REGION Network 38: Sepa Gripper Job Interface [Reloading]
   RUNG wire#powerrail
      Contact( "Unit1.Em7.ControlNodes".sepaGripper."step".action1[421] )
      Coil( "Unit1.Em7.ControlNodes".sepaGripper.jobInterface.reLoadJob4.loadingReady )
   END_RUNG
   RUNG wire#powerrail
      Contact( "Unit1.Em7.ControlNodes".sepaGripper."step".action1[1525] )
      Coil( "Unit1.Em7.ControlNodes".sepaGripper.jobInterface.LoadToJRWinderJob15.loadingReady )
   END_RUNG
   // the same network as SCL:
   "Unit1.Em7.ControlNodes".sepaGripper.jobInterface.reLoadJob4.loadingReady := "Unit1.Em7.ControlNodes".sepaGripper."step".action1[421];
   "Unit1.Em7.ControlNodes".sepaGripper.jobInterface.LoadToJRWinderJob15.loadingReady := "Unit1.Em7.ControlNodes".sepaGripper."step".action1[1525];
END_REGION

REGION Network 39: Sepa Gripper Job Interface [UnReloading]
   RUNG wire#powerrail
      Contact( "Unit1.Em7.ControlNodes".sepaGripper."step".action1[510] )
      Coil( "Unit1.Em7.ControlNodes".sepaGripper.jobInterface.reUnloadJob5.unLoadingReady )
   END_RUNG
   RUNG wire#powerrail
      Contact( #instSepaGripperJellyRollUnGripJob5.jobStatus.active )
      Contact( "Unit1.Em7.ControlNodes".cm.softCam.sepaGripperAxisX.okDisChargePos.inPos )
      Contact( "Unit1.Em7.ControlNodes".cm.softCam.sepaGripperAxisZ.okDisChargePos.inPos )
      Contact( "Unit1.Em7.ControlNodes".cm.softCam.sepaGripperAxisC.okDischargePos.inPos )
      Coil( "Unit1.Em7.ControlNodes".sepaGripper.jobInterface.reUnloadJob5.clampRequest )
   END_RUNG
   RUNG wire#powerrail
      Contact( "Unit1.Em7.ControlNodes".sepaGripper."step".action1[581] )
      Coil( "Unit1.Em7.ControlNodes".sepaGripper.jobInterface.reUnloadJob5.unLoadingDone )
   END_RUNG
   // the same network as SCL:
   "Unit1.Em7.ControlNodes".sepaGripper.jobInterface.reUnloadJob5.unLoadingReady := "Unit1.Em7.ControlNodes".sepaGripper."step".action1[510];
   "Unit1.Em7.ControlNodes".sepaGripper.jobInterface.reUnloadJob5.clampRequest := #instSepaGripperJellyRollUnGripJob5.jobStatus.active AND "Unit1.Em7.ControlNodes".cm.softCam.sepaGripperAxisX.okDisChargePos.inPos AND "Unit1.Em7.ControlNodes".cm.softCam.sepaGripperAxisZ.okDisChargePos.inPos AND "Unit1.Em7.ControlNodes".cm.softCam.sepaGripperAxisC.okDischargePos.inPos;
   "Unit1.Em7.ControlNodes".sepaGripper.jobInterface.reUnloadJob5.unLoadingDone := "Unit1.Em7.ControlNodes".sepaGripper."step".action1[581];
END_REGION

REGION Network 40: [Sepa Gripper Job Interface [UnLoading][BA060]][Unused]
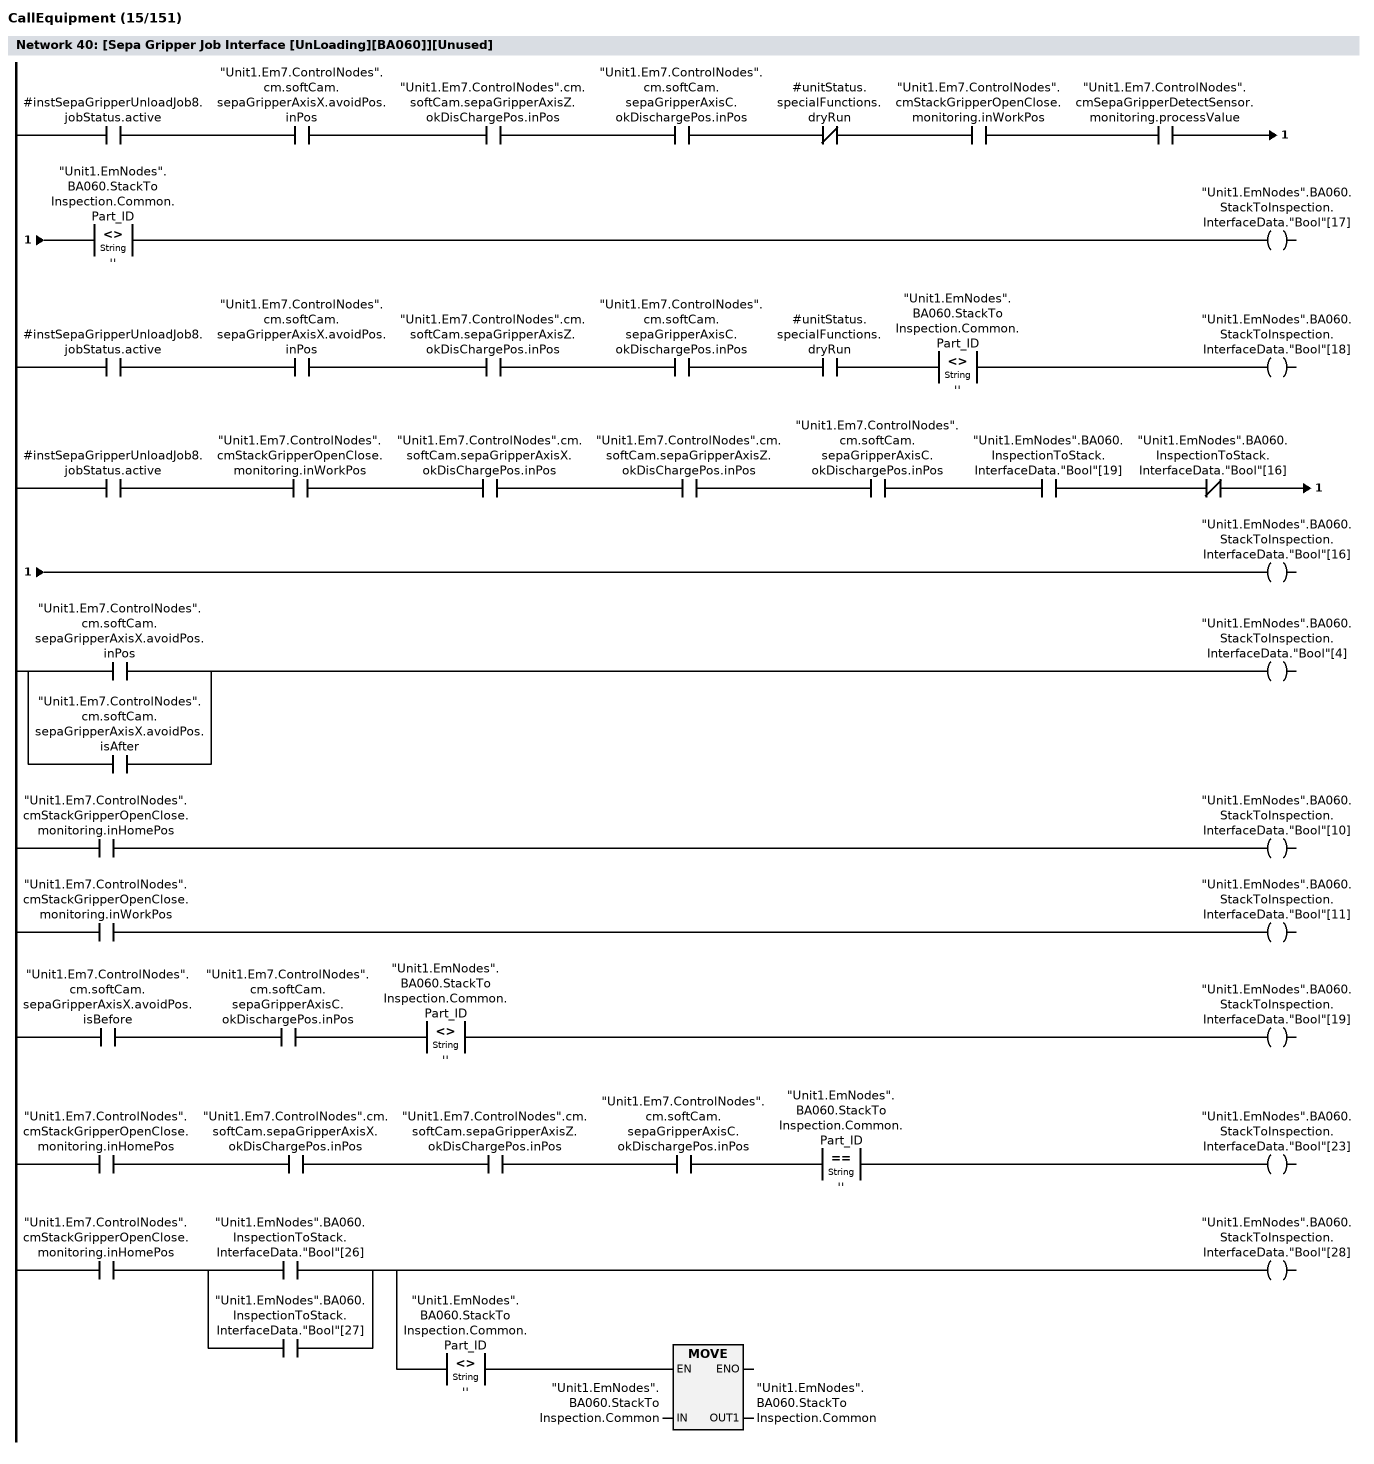
   RUNG wire#powerrail
      Contact( #instSepaGripperUnloadJob8.jobStatus.active )
      Contact( "Unit1.Em7.ControlNodes".cm.softCam.sepaGripperAxisX.avoidPos.inPos )
      Contact( "Unit1.Em7.ControlNodes".cm.softCam.sepaGripperAxisZ.okDisChargePos.inPos )
      Contact( "Unit1.Em7.ControlNodes".cm.softCam.sepaGripperAxisC.okDischargePos.inPos )
      I_Contact( #unitStatus.specialFunctions.dryRun )
      Contact( "Unit1.Em7.ControlNodes".cmStackGripperOpenClose.monitoring.inWorkPos )
      Contact( "Unit1.Em7.ControlNodes".cmSepaGripperDetectSensor.monitoring.processValue )
      { S7_Templates := "SrcType := String" } NE_Contact(in1 := "Unit1.EmNodes".BA060.StackToInspection.Common.Part_ID, in2 := '')
      Coil( "Unit1.EmNodes".BA060.StackToInspection.InterfaceData."Bool"[17] )
   END_RUNG
   RUNG wire#powerrail
      Contact( #instSepaGripperUnloadJob8.jobStatus.active )
      Contact( "Unit1.Em7.ControlNodes".cm.softCam.sepaGripperAxisX.avoidPos.inPos )
      Contact( "Unit1.Em7.ControlNodes".cm.softCam.sepaGripperAxisZ.okDisChargePos.inPos )
      Contact( "Unit1.Em7.ControlNodes".cm.softCam.sepaGripperAxisC.okDischargePos.inPos )
      Contact( #unitStatus.specialFunctions.dryRun )
      { S7_Templates := "SrcType := String" } NE_Contact(in1 := "Unit1.EmNodes".BA060.StackToInspection.Common.Part_ID, in2 := '')
      Coil( "Unit1.EmNodes".BA060.StackToInspection.InterfaceData."Bool"[18] )
   END_RUNG
   RUNG wire#powerrail
      Contact( #instSepaGripperUnloadJob8.jobStatus.active )
      Contact( "Unit1.Em7.ControlNodes".cmStackGripperOpenClose.monitoring.inWorkPos )
      Contact( "Unit1.Em7.ControlNodes".cm.softCam.sepaGripperAxisX.okDisChargePos.inPos )
      Contact( "Unit1.Em7.ControlNodes".cm.softCam.sepaGripperAxisZ.okDisChargePos.inPos )
      Contact( "Unit1.Em7.ControlNodes".cm.softCam.sepaGripperAxisC.okDischargePos.inPos )
      Contact( "Unit1.EmNodes".BA060.InspectionToStack.InterfaceData."Bool"[19] )
      I_Contact( "Unit1.EmNodes".BA060.InspectionToStack.InterfaceData."Bool"[16] )
      Coil( "Unit1.EmNodes".BA060.StackToInspection.InterfaceData."Bool"[16] )
   END_RUNG
   RUNG wire#powerrail
      Contact( "Unit1.Em7.ControlNodes".cm.softCam.sepaGripperAxisX.avoidPos.inPos )
      wire#w1
      Coil( "Unit1.EmNodes".BA060.StackToInspection.InterfaceData."Bool"[4] )
   END_RUNG
   RUNG wire#powerrail
      Contact( "Unit1.Em7.ControlNodes".cm.softCam.sepaGripperAxisX.avoidPos.isAfter )
   END_RUNG wire#w1
   RUNG wire#powerrail
      Contact( "Unit1.Em7.ControlNodes".cmStackGripperOpenClose.monitoring.inHomePos )
      Coil( "Unit1.EmNodes".BA060.StackToInspection.InterfaceData."Bool"[10] )
   END_RUNG
   RUNG wire#powerrail
      Contact( "Unit1.Em7.ControlNodes".cmStackGripperOpenClose.monitoring.inWorkPos )
      Coil( "Unit1.EmNodes".BA060.StackToInspection.InterfaceData."Bool"[11] )
   END_RUNG
   RUNG wire#powerrail
      Contact( "Unit1.Em7.ControlNodes".cm.softCam.sepaGripperAxisX.avoidPos.isBefore )
      Contact( "Unit1.Em7.ControlNodes".cm.softCam.sepaGripperAxisC.okDischargePos.inPos )
      { S7_Templates := "SrcType := String" } NE_Contact(in1 := "Unit1.EmNodes".BA060.StackToInspection.Common.Part_ID, in2 := '')
      Coil( "Unit1.EmNodes".BA060.StackToInspection.InterfaceData."Bool"[19] )
   END_RUNG
   RUNG wire#powerrail
      Contact( "Unit1.Em7.ControlNodes".cmStackGripperOpenClose.monitoring.inHomePos )
      Contact( "Unit1.Em7.ControlNodes".cm.softCam.sepaGripperAxisX.okDisChargePos.inPos )
      Contact( "Unit1.Em7.ControlNodes".cm.softCam.sepaGripperAxisZ.okDisChargePos.inPos )
      Contact( "Unit1.Em7.ControlNodes".cm.softCam.sepaGripperAxisC.okDischargePos.inPos )
      { S7_Templates := "SrcType := String" } EQ_Contact(in1 := "Unit1.EmNodes".BA060.StackToInspection.Common.Part_ID, in2 := '')
      Coil( "Unit1.EmNodes".BA060.StackToInspection.InterfaceData."Bool"[23] )
   END_RUNG
   RUNG wire#powerrail
      Contact( "Unit1.Em7.ControlNodes".cmStackGripperOpenClose.monitoring.inHomePos )
      wire#w2
      Contact( "Unit1.EmNodes".BA060.InspectionToStack.InterfaceData."Bool"[26] )
      wire#w3
      Coil( "Unit1.EmNodes".BA060.StackToInspection.InterfaceData."Bool"[28] )
   END_RUNG
   RUNG wire#w2
      Contact( "Unit1.EmNodes".BA060.InspectionToStack.InterfaceData."Bool"[27] )
   END_RUNG wire#w3
   RUNG wire#w3
      { S7_Templates := "SrcType := String" } NE_Contact(in1 := "Unit1.EmNodes".BA060.StackToInspection.Common.Part_ID, in2 := '')
      Move(in := "Unit1.EmNodes".BA060.StackToInspection.Common, out1 => "Unit1.EmNodes".BA060.StackToInspection.Common)
   END_RUNG
   // the same network as SCL:
   "Unit1.EmNodes".BA060.StackToInspection.InterfaceData."Bool"[17] := #instSepaGripperUnloadJob8.jobStatus.active AND "Unit1.Em7.ControlNodes".cm.softCam.sepaGripperAxisX.avoidPos.inPos AND "Unit1.Em7.ControlNodes".cm.softCam.sepaGripperAxisZ.okDisChargePos.inPos AND "Unit1.Em7.ControlNodes".cm.softCam.sepaGripperAxisC.okDischargePos.inPos AND NOT #unitStatus.specialFunctions.dryRun AND "Unit1.Em7.ControlNodes".cmStackGripperOpenClose.monitoring.inWorkPos AND "Unit1.Em7.ControlNodes".cmSepaGripperDetectSensor.monitoring.processValue AND ("Unit1.EmNodes".BA060.StackToInspection.Common.Part_ID <> '');
   "Unit1.EmNodes".BA060.StackToInspection.InterfaceData."Bool"[18] := #instSepaGripperUnloadJob8.jobStatus.active AND "Unit1.Em7.ControlNodes".cm.softCam.sepaGripperAxisX.avoidPos.inPos AND "Unit1.Em7.ControlNodes".cm.softCam.sepaGripperAxisZ.okDisChargePos.inPos AND "Unit1.Em7.ControlNodes".cm.softCam.sepaGripperAxisC.okDischargePos.inPos AND #unitStatus.specialFunctions.dryRun AND ("Unit1.EmNodes".BA060.StackToInspection.Common.Part_ID <> '');
   "Unit1.EmNodes".BA060.StackToInspection.InterfaceData."Bool"[16] := #instSepaGripperUnloadJob8.jobStatus.active AND "Unit1.Em7.ControlNodes".cmStackGripperOpenClose.monitoring.inWorkPos AND "Unit1.Em7.ControlNodes".cm.softCam.sepaGripperAxisX.okDisChargePos.inPos AND "Unit1.Em7.ControlNodes".cm.softCam.sepaGripperAxisZ.okDisChargePos.inPos AND "Unit1.Em7.ControlNodes".cm.softCam.sepaGripperAxisC.okDischargePos.inPos AND "Unit1.EmNodes".BA060.InspectionToStack.InterfaceData."Bool"[19] AND NOT "Unit1.EmNodes".BA060.InspectionToStack.InterfaceData."Bool"[16];
   "Unit1.EmNodes".BA060.StackToInspection.InterfaceData."Bool"[4] := "Unit1.Em7.ControlNodes".cm.softCam.sepaGripperAxisX.avoidPos.inPos OR "Unit1.Em7.ControlNodes".cm.softCam.sepaGripperAxisX.avoidPos.isAfter;
   "Unit1.EmNodes".BA060.StackToInspection.InterfaceData."Bool"[10] := "Unit1.Em7.ControlNodes".cmStackGripperOpenClose.monitoring.inHomePos;
   "Unit1.EmNodes".BA060.StackToInspection.InterfaceData."Bool"[11] := "Unit1.Em7.ControlNodes".cmStackGripperOpenClose.monitoring.inWorkPos;
   "Unit1.EmNodes".BA060.StackToInspection.InterfaceData."Bool"[19] := "Unit1.Em7.ControlNodes".cm.softCam.sepaGripperAxisX.avoidPos.isBefore AND "Unit1.Em7.ControlNodes".cm.softCam.sepaGripperAxisC.okDischargePos.inPos AND ("Unit1.EmNodes".BA060.StackToInspection.Common.Part_ID <> '');
   "Unit1.EmNodes".BA060.StackToInspection.InterfaceData."Bool"[23] := "Unit1.Em7.ControlNodes".cmStackGripperOpenClose.monitoring.inHomePos AND "Unit1.Em7.ControlNodes".cm.softCam.sepaGripperAxisX.okDisChargePos.inPos AND "Unit1.Em7.ControlNodes".cm.softCam.sepaGripperAxisZ.okDisChargePos.inPos AND "Unit1.Em7.ControlNodes".cm.softCam.sepaGripperAxisC.okDischargePos.inPos AND ("Unit1.EmNodes".BA060.StackToInspection.Common.Part_ID = '');
   "Unit1.EmNodes".BA060.StackToInspection.InterfaceData."Bool"[28] := "Unit1.Em7.ControlNodes".cmStackGripperOpenClose.monitoring.inHomePos AND ("Unit1.EmNodes".BA060.InspectionToStack.InterfaceData."Bool"[26] OR "Unit1.EmNodes".BA060.InspectionToStack.InterfaceData."Bool"[27]);
   IF "Unit1.Em7.ControlNodes".cmStackGripperOpenClose.monitoring.inHomePos AND ("Unit1.EmNodes".BA060.InspectionToStack.InterfaceData."Bool"[26] OR "Unit1.EmNodes".BA060.InspectionToStack.InterfaceData."Bool"[27]) AND ("Unit1.EmNodes".BA060.StackToInspection.Common.Part_ID <> '') THEN
       "Unit1.EmNodes".BA060.StackToInspection.Common := "Unit1.EmNodes".BA060.StackToInspection.Common;
   END_IF;
END_REGION

REGION Network 41: Sepa Gripper Job Interface Working Done
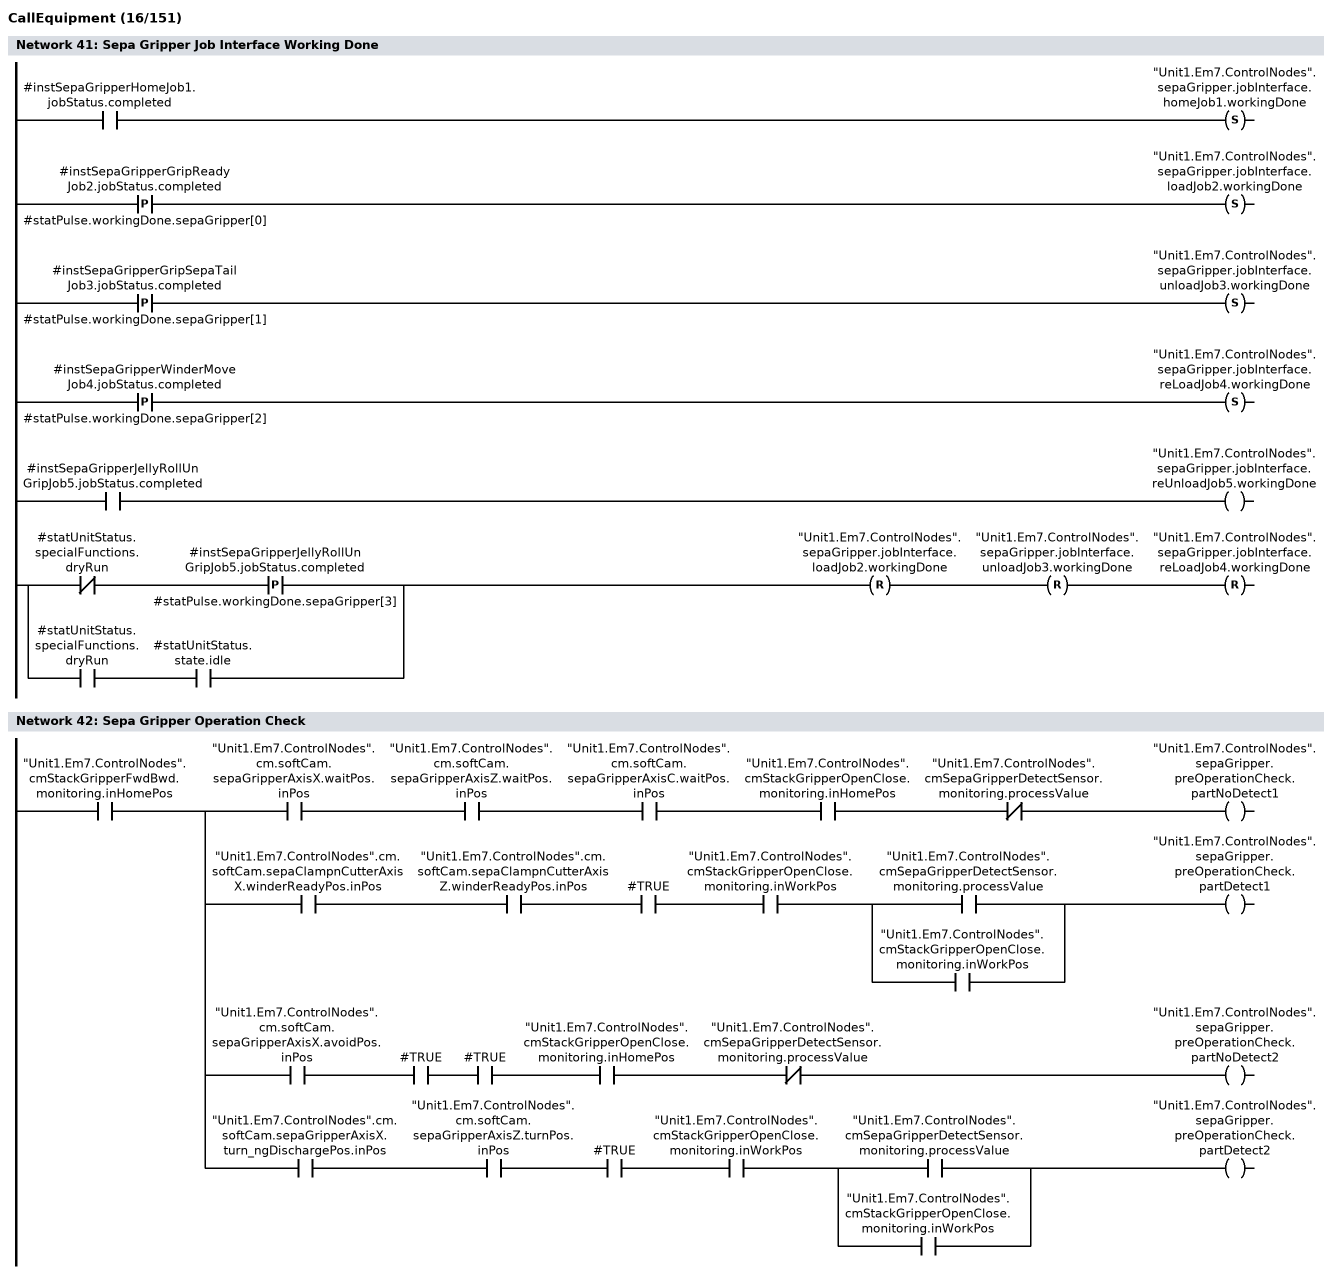
   RUNG wire#powerrail
      Contact( #instSepaGripperHomeJob1.jobStatus.completed )
      S_Coil( "Unit1.Em7.ControlNodes".sepaGripper.jobInterface.homeJob1.workingDone )
   END_RUNG
   RUNG wire#powerrail
      P_Contact(operand := #instSepaGripperGripReadyJob2.jobStatus.completed, bit := #statPulse.workingDone.sepaGripper[0])
      S_Coil( "Unit1.Em7.ControlNodes".sepaGripper.jobInterface.loadJob2.workingDone )
   END_RUNG
   RUNG wire#powerrail
      P_Contact(operand := #instSepaGripperGripSepaTailJob3.jobStatus.completed, bit := #statPulse.workingDone.sepaGripper[1])
      S_Coil( "Unit1.Em7.ControlNodes".sepaGripper.jobInterface.unloadJob3.workingDone )
   END_RUNG
   RUNG wire#powerrail
      P_Contact(operand := #instSepaGripperWinderMoveJob4.jobStatus.completed, bit := #statPulse.workingDone.sepaGripper[2])
      S_Coil( "Unit1.Em7.ControlNodes".sepaGripper.jobInterface.reLoadJob4.workingDone )
   END_RUNG
   RUNG wire#powerrail
      Contact( #instSepaGripperJellyRollUnGripJob5.jobStatus.completed )
      Coil( "Unit1.Em7.ControlNodes".sepaGripper.jobInterface.reUnloadJob5.workingDone )
   END_RUNG
   RUNG wire#powerrail
      I_Contact( #statUnitStatus.specialFunctions.dryRun )
      P_Contact(operand := #instSepaGripperJellyRollUnGripJob5.jobStatus.completed, bit := #statPulse.workingDone.sepaGripper[3])
      wire#w1
      R_Coil( "Unit1.Em7.ControlNodes".sepaGripper.jobInterface.loadJob2.workingDone )
      R_Coil( "Unit1.Em7.ControlNodes".sepaGripper.jobInterface.unloadJob3.workingDone )
      R_Coil( "Unit1.Em7.ControlNodes".sepaGripper.jobInterface.reLoadJob4.workingDone )
   END_RUNG
   RUNG wire#powerrail
      Contact( #statUnitStatus.specialFunctions.dryRun )
      Contact( #statUnitStatus.state.idle )
   END_RUNG wire#w1
   // the same network as SCL:
   IF #instSepaGripperHomeJob1.jobStatus.completed THEN
       "Unit1.Em7.ControlNodes".sepaGripper.jobInterface.homeJob1.workingDone := TRUE;
   END_IF;
   #_w1 := #instSepaGripperGripReadyJob2.jobStatus.completed AND NOT #statPulse.workingDone.sepaGripper[0];   // rising edge of #instSepaGripperGripReadyJob2.jobStatus.completed
   #statPulse.workingDone.sepaGripper[0] := #instSepaGripperGripReadyJob2.jobStatus.completed;
   IF #_w1 THEN "Unit1.Em7.ControlNodes".sepaGripper.jobInterface.loadJob2.workingDone := TRUE; END_IF;
   #_w2 := #instSepaGripperGripSepaTailJob3.jobStatus.completed AND NOT #statPulse.workingDone.sepaGripper[1];   // rising edge of #instSepaGripperGripSepaTailJob3.jobStatus.completed
   #statPulse.workingDone.sepaGripper[1] := #instSepaGripperGripSepaTailJob3.jobStatus.completed;
   IF #_w2 THEN "Unit1.Em7.ControlNodes".sepaGripper.jobInterface.unloadJob3.workingDone := TRUE; END_IF;
   #_w3 := #instSepaGripperWinderMoveJob4.jobStatus.completed AND NOT #statPulse.workingDone.sepaGripper[2];   // rising edge of #instSepaGripperWinderMoveJob4.jobStatus.completed
   #statPulse.workingDone.sepaGripper[2] := #instSepaGripperWinderMoveJob4.jobStatus.completed;
   IF #_w3 THEN "Unit1.Em7.ControlNodes".sepaGripper.jobInterface.reLoadJob4.workingDone := TRUE; END_IF;
   "Unit1.Em7.ControlNodes".sepaGripper.jobInterface.reUnloadJob5.workingDone := #instSepaGripperJellyRollUnGripJob5.jobStatus.completed;
   #_w4 := NOT #statUnitStatus.specialFunctions.dryRun AND #instSepaGripperJellyRollUnGripJob5.jobStatus.completed AND NOT #statPulse.workingDone.sepaGripper[3];   // rising edge of #instSepaGripperJellyRollUnGripJob5.jobStatus.completed
   #statPulse.workingDone.sepaGripper[3] := #instSepaGripperJellyRollUnGripJob5.jobStatus.completed;
   IF #_w4 OR (#statUnitStatus.specialFunctions.dryRun AND #statUnitStatus.state.idle) THEN
       "Unit1.Em7.ControlNodes".sepaGripper.jobInterface.loadJob2.workingDone := FALSE;
       "Unit1.Em7.ControlNodes".sepaGripper.jobInterface.unloadJob3.workingDone := FALSE;
       "Unit1.Em7.ControlNodes".sepaGripper.jobInterface.reLoadJob4.workingDone := FALSE;
   END_IF;
END_REGION

REGION Network 42: Sepa Gripper Operation Check
   RUNG wire#powerrail
      Contact( "Unit1.Em7.ControlNodes".cmStackGripperFwdBwd.monitoring.inHomePos )
      wire#w1
      Contact( "Unit1.Em7.ControlNodes".cm.softCam.sepaGripperAxisX.waitPos.inPos )
      Contact( "Unit1.Em7.ControlNodes".cm.softCam.sepaGripperAxisZ.waitPos.inPos )
      Contact( "Unit1.Em7.ControlNodes".cm.softCam.sepaGripperAxisC.waitPos.inPos )
      Contact( "Unit1.Em7.ControlNodes".cmStackGripperOpenClose.monitoring.inHomePos )
      I_Contact( "Unit1.Em7.ControlNodes".cmSepaGripperDetectSensor.monitoring.processValue )
      Coil( "Unit1.Em7.ControlNodes".sepaGripper.preOperationCheck.partNoDetect1 )
   END_RUNG
   RUNG wire#w1
      Contact( "Unit1.Em7.ControlNodes".cm.softCam.sepaClampnCutterAxisX.winderReadyPos.inPos )
      Contact( "Unit1.Em7.ControlNodes".cm.softCam.sepaClampnCutterAxisZ.winderReadyPos.inPos )
      Contact( #TRUE )
      Contact( "Unit1.Em7.ControlNodes".cmStackGripperOpenClose.monitoring.inWorkPos )
      wire#w2
      Contact( "Unit1.Em7.ControlNodes".cmSepaGripperDetectSensor.monitoring.processValue )
      wire#w3
      Coil( "Unit1.Em7.ControlNodes".sepaGripper.preOperationCheck.partDetect1 )
   END_RUNG
   RUNG wire#w2
      Contact( "Unit1.Em7.ControlNodes".cmStackGripperOpenClose.monitoring.inWorkPos )
   END_RUNG wire#w3
   RUNG wire#w1
      Contact( "Unit1.Em7.ControlNodes".cm.softCam.sepaGripperAxisX.avoidPos.inPos )
      Contact( #TRUE )
      Contact( #TRUE )
      Contact( "Unit1.Em7.ControlNodes".cmStackGripperOpenClose.monitoring.inHomePos )
      I_Contact( "Unit1.Em7.ControlNodes".cmSepaGripperDetectSensor.monitoring.processValue )
      Coil( "Unit1.Em7.ControlNodes".sepaGripper.preOperationCheck.partNoDetect2 )
   END_RUNG
   RUNG wire#w1
      Contact( "Unit1.Em7.ControlNodes".cm.softCam.sepaGripperAxisX.turn_ngDischargePos.inPos )
      Contact( "Unit1.Em7.ControlNodes".cm.softCam.sepaGripperAxisZ.turnPos.inPos )
      Contact( #TRUE )
      Contact( "Unit1.Em7.ControlNodes".cmStackGripperOpenClose.monitoring.inWorkPos )
      wire#w4
      Contact( "Unit1.Em7.ControlNodes".cmSepaGripperDetectSensor.monitoring.processValue )
      wire#w5
      Coil( "Unit1.Em7.ControlNodes".sepaGripper.preOperationCheck.partDetect2 )
   END_RUNG
   RUNG wire#w4
      Contact( "Unit1.Em7.ControlNodes".cmStackGripperOpenClose.monitoring.inWorkPos )
   END_RUNG wire#w5
   // the same network as SCL:
   "Unit1.Em7.ControlNodes".sepaGripper.preOperationCheck.partNoDetect1 := "Unit1.Em7.ControlNodes".cmStackGripperFwdBwd.monitoring.inHomePos AND "Unit1.Em7.ControlNodes".cm.softCam.sepaGripperAxisX.waitPos.inPos AND "Unit1.Em7.ControlNodes".cm.softCam.sepaGripperAxisZ.waitPos.inPos AND "Unit1.Em7.ControlNodes".cm.softCam.sepaGripperAxisC.waitPos.inPos AND "Unit1.Em7.ControlNodes".cmStackGripperOpenClose.monitoring.inHomePos AND NOT "Unit1.Em7.ControlNodes".cmSepaGripperDetectSensor.monitoring.processValue;
   "Unit1.Em7.ControlNodes".sepaGripper.preOperationCheck.partDetect1 := "Unit1.Em7.ControlNodes".cmStackGripperFwdBwd.monitoring.inHomePos AND "Unit1.Em7.ControlNodes".cm.softCam.sepaClampnCutterAxisX.winderReadyPos.inPos AND "Unit1.Em7.ControlNodes".cm.softCam.sepaClampnCutterAxisZ.winderReadyPos.inPos AND #TRUE AND "Unit1.Em7.ControlNodes".cmStackGripperOpenClose.monitoring.inWorkPos AND ("Unit1.Em7.ControlNodes".cmSepaGripperDetectSensor.monitoring.processValue OR "Unit1.Em7.ControlNodes".cmStackGripperOpenClose.monitoring.inWorkPos);
   "Unit1.Em7.ControlNodes".sepaGripper.preOperationCheck.partNoDetect2 := "Unit1.Em7.ControlNodes".cmStackGripperFwdBwd.monitoring.inHomePos AND "Unit1.Em7.ControlNodes".cm.softCam.sepaGripperAxisX.avoidPos.inPos AND #TRUE AND #TRUE AND "Unit1.Em7.ControlNodes".cmStackGripperOpenClose.monitoring.inHomePos AND NOT "Unit1.Em7.ControlNodes".cmSepaGripperDetectSensor.monitoring.processValue;
   "Unit1.Em7.ControlNodes".sepaGripper.preOperationCheck.partDetect2 := "Unit1.Em7.ControlNodes".cmStackGripperFwdBwd.monitoring.inHomePos AND "Unit1.Em7.ControlNodes".cm.softCam.sepaGripperAxisX.turn_ngDischargePos.inPos AND "Unit1.Em7.ControlNodes".cm.softCam.sepaGripperAxisZ.turnPos.inPos AND #TRUE AND "Unit1.Em7.ControlNodes".cmStackGripperOpenClose.monitoring.inWorkPos AND ("Unit1.Em7.ControlNodes".cmSepaGripperDetectSensor.monitoring.processValue OR "Unit1.Em7.ControlNodes".cmStackGripperOpenClose.monitoring.inWorkPos);
END_REGION

REGION Network 43: Sepa Gripper Operation Check [Cam]
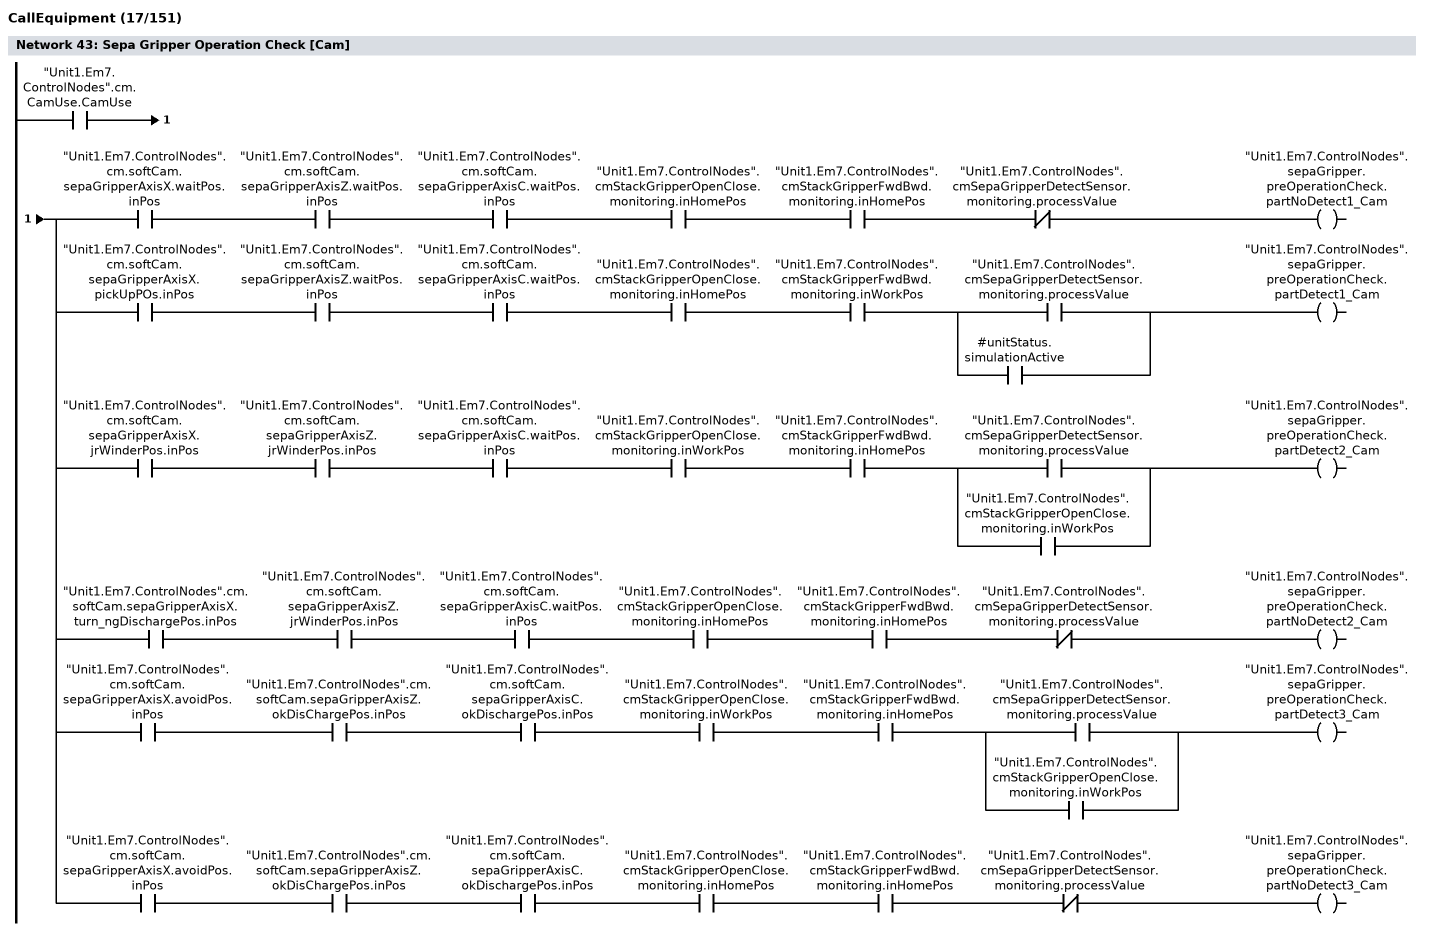
   RUNG wire#powerrail
      Contact( "Unit1.Em7.ControlNodes".cm.CamUse.CamUse )
      wire#w1
      Contact( "Unit1.Em7.ControlNodes".cm.softCam.sepaGripperAxisX.waitPos.inPos )
      Contact( "Unit1.Em7.ControlNodes".cm.softCam.sepaGripperAxisZ.waitPos.inPos )
      Contact( "Unit1.Em7.ControlNodes".cm.softCam.sepaGripperAxisC.waitPos.inPos )
      Contact( "Unit1.Em7.ControlNodes".cmStackGripperOpenClose.monitoring.inHomePos )
      Contact( "Unit1.Em7.ControlNodes".cmStackGripperFwdBwd.monitoring.inHomePos )
      I_Contact( "Unit1.Em7.ControlNodes".cmSepaGripperDetectSensor.monitoring.processValue )
      Coil( "Unit1.Em7.ControlNodes".sepaGripper.preOperationCheck.partNoDetect1_Cam )
   END_RUNG
   RUNG wire#w1
      Contact( "Unit1.Em7.ControlNodes".cm.softCam.sepaGripperAxisX.pickUpPOs.inPos )
      Contact( "Unit1.Em7.ControlNodes".cm.softCam.sepaGripperAxisZ.waitPos.inPos )
      Contact( "Unit1.Em7.ControlNodes".cm.softCam.sepaGripperAxisC.waitPos.inPos )
      Contact( "Unit1.Em7.ControlNodes".cmStackGripperOpenClose.monitoring.inHomePos )
      Contact( "Unit1.Em7.ControlNodes".cmStackGripperFwdBwd.monitoring.inWorkPos )
      wire#w2
      Contact( "Unit1.Em7.ControlNodes".cmSepaGripperDetectSensor.monitoring.processValue )
      wire#w3
      Coil( "Unit1.Em7.ControlNodes".sepaGripper.preOperationCheck.partDetect1_Cam )
   END_RUNG
   RUNG wire#w2
      Contact( #unitStatus.simulationActive )
   END_RUNG wire#w3
   RUNG wire#w1
      Contact( "Unit1.Em7.ControlNodes".cm.softCam.sepaGripperAxisX.jrWinderPos.inPos )
      Contact( "Unit1.Em7.ControlNodes".cm.softCam.sepaGripperAxisZ.jrWinderPos.inPos )
      Contact( "Unit1.Em7.ControlNodes".cm.softCam.sepaGripperAxisC.waitPos.inPos )
      Contact( "Unit1.Em7.ControlNodes".cmStackGripperOpenClose.monitoring.inWorkPos )
      Contact( "Unit1.Em7.ControlNodes".cmStackGripperFwdBwd.monitoring.inHomePos )
      wire#w4
      Contact( "Unit1.Em7.ControlNodes".cmSepaGripperDetectSensor.monitoring.processValue )
      wire#w5
      Coil( "Unit1.Em7.ControlNodes".sepaGripper.preOperationCheck.partDetect2_Cam )
   END_RUNG
   RUNG wire#w4
      Contact( "Unit1.Em7.ControlNodes".cmStackGripperOpenClose.monitoring.inWorkPos )
   END_RUNG wire#w5
   RUNG wire#w1
      Contact( "Unit1.Em7.ControlNodes".cm.softCam.sepaGripperAxisX.turn_ngDischargePos.inPos )
      Contact( "Unit1.Em7.ControlNodes".cm.softCam.sepaGripperAxisZ.jrWinderPos.inPos )
      Contact( "Unit1.Em7.ControlNodes".cm.softCam.sepaGripperAxisC.waitPos.inPos )
      Contact( "Unit1.Em7.ControlNodes".cmStackGripperOpenClose.monitoring.inHomePos )
      Contact( "Unit1.Em7.ControlNodes".cmStackGripperFwdBwd.monitoring.inHomePos )
      I_Contact( "Unit1.Em7.ControlNodes".cmSepaGripperDetectSensor.monitoring.processValue )
      Coil( "Unit1.Em7.ControlNodes".sepaGripper.preOperationCheck.partNoDetect2_Cam )
   END_RUNG
   RUNG wire#w1
      Contact( "Unit1.Em7.ControlNodes".cm.softCam.sepaGripperAxisX.avoidPos.inPos )
      Contact( "Unit1.Em7.ControlNodes".cm.softCam.sepaGripperAxisZ.okDisChargePos.inPos )
      Contact( "Unit1.Em7.ControlNodes".cm.softCam.sepaGripperAxisC.okDischargePos.inPos )
      Contact( "Unit1.Em7.ControlNodes".cmStackGripperOpenClose.monitoring.inWorkPos )
      Contact( "Unit1.Em7.ControlNodes".cmStackGripperFwdBwd.monitoring.inHomePos )
      wire#w6
      Contact( "Unit1.Em7.ControlNodes".cmSepaGripperDetectSensor.monitoring.processValue )
      wire#w7
      Coil( "Unit1.Em7.ControlNodes".sepaGripper.preOperationCheck.partDetect3_Cam )
   END_RUNG
   RUNG wire#w6
      Contact( "Unit1.Em7.ControlNodes".cmStackGripperOpenClose.monitoring.inWorkPos )
   END_RUNG wire#w7
   RUNG wire#w1
      Contact( "Unit1.Em7.ControlNodes".cm.softCam.sepaGripperAxisX.avoidPos.inPos )
      Contact( "Unit1.Em7.ControlNodes".cm.softCam.sepaGripperAxisZ.okDisChargePos.inPos )
      Contact( "Unit1.Em7.ControlNodes".cm.softCam.sepaGripperAxisC.okDischargePos.inPos )
      Contact( "Unit1.Em7.ControlNodes".cmStackGripperOpenClose.monitoring.inHomePos )
      Contact( "Unit1.Em7.ControlNodes".cmStackGripperFwdBwd.monitoring.inHomePos )
      I_Contact( "Unit1.Em7.ControlNodes".cmSepaGripperDetectSensor.monitoring.processValue )
      Coil( "Unit1.Em7.ControlNodes".sepaGripper.preOperationCheck.partNoDetect3_Cam )
   END_RUNG
   // the same network as SCL:
   "Unit1.Em7.ControlNodes".sepaGripper.preOperationCheck.partNoDetect1_Cam := "Unit1.Em7.ControlNodes".cm.CamUse.CamUse AND "Unit1.Em7.ControlNodes".cm.softCam.sepaGripperAxisX.waitPos.inPos AND "Unit1.Em7.ControlNodes".cm.softCam.sepaGripperAxisZ.waitPos.inPos AND "Unit1.Em7.ControlNodes".cm.softCam.sepaGripperAxisC.waitPos.inPos AND "Unit1.Em7.ControlNodes".cmStackGripperOpenClose.monitoring.inHomePos AND "Unit1.Em7.ControlNodes".cmStackGripperFwdBwd.monitoring.inHomePos AND NOT "Unit1.Em7.ControlNodes".cmSepaGripperDetectSensor.monitoring.processValue;
   "Unit1.Em7.ControlNodes".sepaGripper.preOperationCheck.partDetect1_Cam := "Unit1.Em7.ControlNodes".cm.CamUse.CamUse AND "Unit1.Em7.ControlNodes".cm.softCam.sepaGripperAxisX.pickUpPOs.inPos AND "Unit1.Em7.ControlNodes".cm.softCam.sepaGripperAxisZ.waitPos.inPos AND "Unit1.Em7.ControlNodes".cm.softCam.sepaGripperAxisC.waitPos.inPos AND "Unit1.Em7.ControlNodes".cmStackGripperOpenClose.monitoring.inHomePos AND "Unit1.Em7.ControlNodes".cmStackGripperFwdBwd.monitoring.inWorkPos AND ("Unit1.Em7.ControlNodes".cmSepaGripperDetectSensor.monitoring.processValue OR #unitStatus.simulationActive);
   "Unit1.Em7.ControlNodes".sepaGripper.preOperationCheck.partDetect2_Cam := "Unit1.Em7.ControlNodes".cm.CamUse.CamUse AND "Unit1.Em7.ControlNodes".cm.softCam.sepaGripperAxisX.jrWinderPos.inPos AND "Unit1.Em7.ControlNodes".cm.softCam.sepaGripperAxisZ.jrWinderPos.inPos AND "Unit1.Em7.ControlNodes".cm.softCam.sepaGripperAxisC.waitPos.inPos AND "Unit1.Em7.ControlNodes".cmStackGripperOpenClose.monitoring.inWorkPos AND "Unit1.Em7.ControlNodes".cmStackGripperFwdBwd.monitoring.inHomePos AND ("Unit1.Em7.ControlNodes".cmSepaGripperDetectSensor.monitoring.processValue OR "Unit1.Em7.ControlNodes".cmStackGripperOpenClose.monitoring.inWorkPos);
   "Unit1.Em7.ControlNodes".sepaGripper.preOperationCheck.partNoDetect2_Cam := "Unit1.Em7.ControlNodes".cm.CamUse.CamUse AND "Unit1.Em7.ControlNodes".cm.softCam.sepaGripperAxisX.turn_ngDischargePos.inPos AND "Unit1.Em7.ControlNodes".cm.softCam.sepaGripperAxisZ.jrWinderPos.inPos AND "Unit1.Em7.ControlNodes".cm.softCam.sepaGripperAxisC.waitPos.inPos AND "Unit1.Em7.ControlNodes".cmStackGripperOpenClose.monitoring.inHomePos AND "Unit1.Em7.ControlNodes".cmStackGripperFwdBwd.monitoring.inHomePos AND NOT "Unit1.Em7.ControlNodes".cmSepaGripperDetectSensor.monitoring.processValue;
   "Unit1.Em7.ControlNodes".sepaGripper.preOperationCheck.partDetect3_Cam := "Unit1.Em7.ControlNodes".cm.CamUse.CamUse AND "Unit1.Em7.ControlNodes".cm.softCam.sepaGripperAxisX.avoidPos.inPos AND "Unit1.Em7.ControlNodes".cm.softCam.sepaGripperAxisZ.okDisChargePos.inPos AND "Unit1.Em7.ControlNodes".cm.softCam.sepaGripperAxisC.okDischargePos.inPos AND "Unit1.Em7.ControlNodes".cmStackGripperOpenClose.monitoring.inWorkPos AND "Unit1.Em7.ControlNodes".cmStackGripperFwdBwd.monitoring.inHomePos AND ("Unit1.Em7.ControlNodes".cmSepaGripperDetectSensor.monitoring.processValue OR "Unit1.Em7.ControlNodes".cmStackGripperOpenClose.monitoring.inWorkPos);
   "Unit1.Em7.ControlNodes".sepaGripper.preOperationCheck.partNoDetect3_Cam := "Unit1.Em7.ControlNodes".cm.CamUse.CamUse AND "Unit1.Em7.ControlNodes".cm.softCam.sepaGripperAxisX.avoidPos.inPos AND "Unit1.Em7.ControlNodes".cm.softCam.sepaGripperAxisZ.okDisChargePos.inPos AND "Unit1.Em7.ControlNodes".cm.softCam.sepaGripperAxisC.okDischargePos.inPos AND "Unit1.Em7.ControlNodes".cmStackGripperOpenClose.monitoring.inHomePos AND "Unit1.Em7.ControlNodes".cmStackGripperFwdBwd.monitoring.inHomePos AND NOT "Unit1.Em7.ControlNodes".cmSepaGripperDetectSensor.monitoring.processValue;
END_REGION

REGION Network 45: JR Winder Select Job
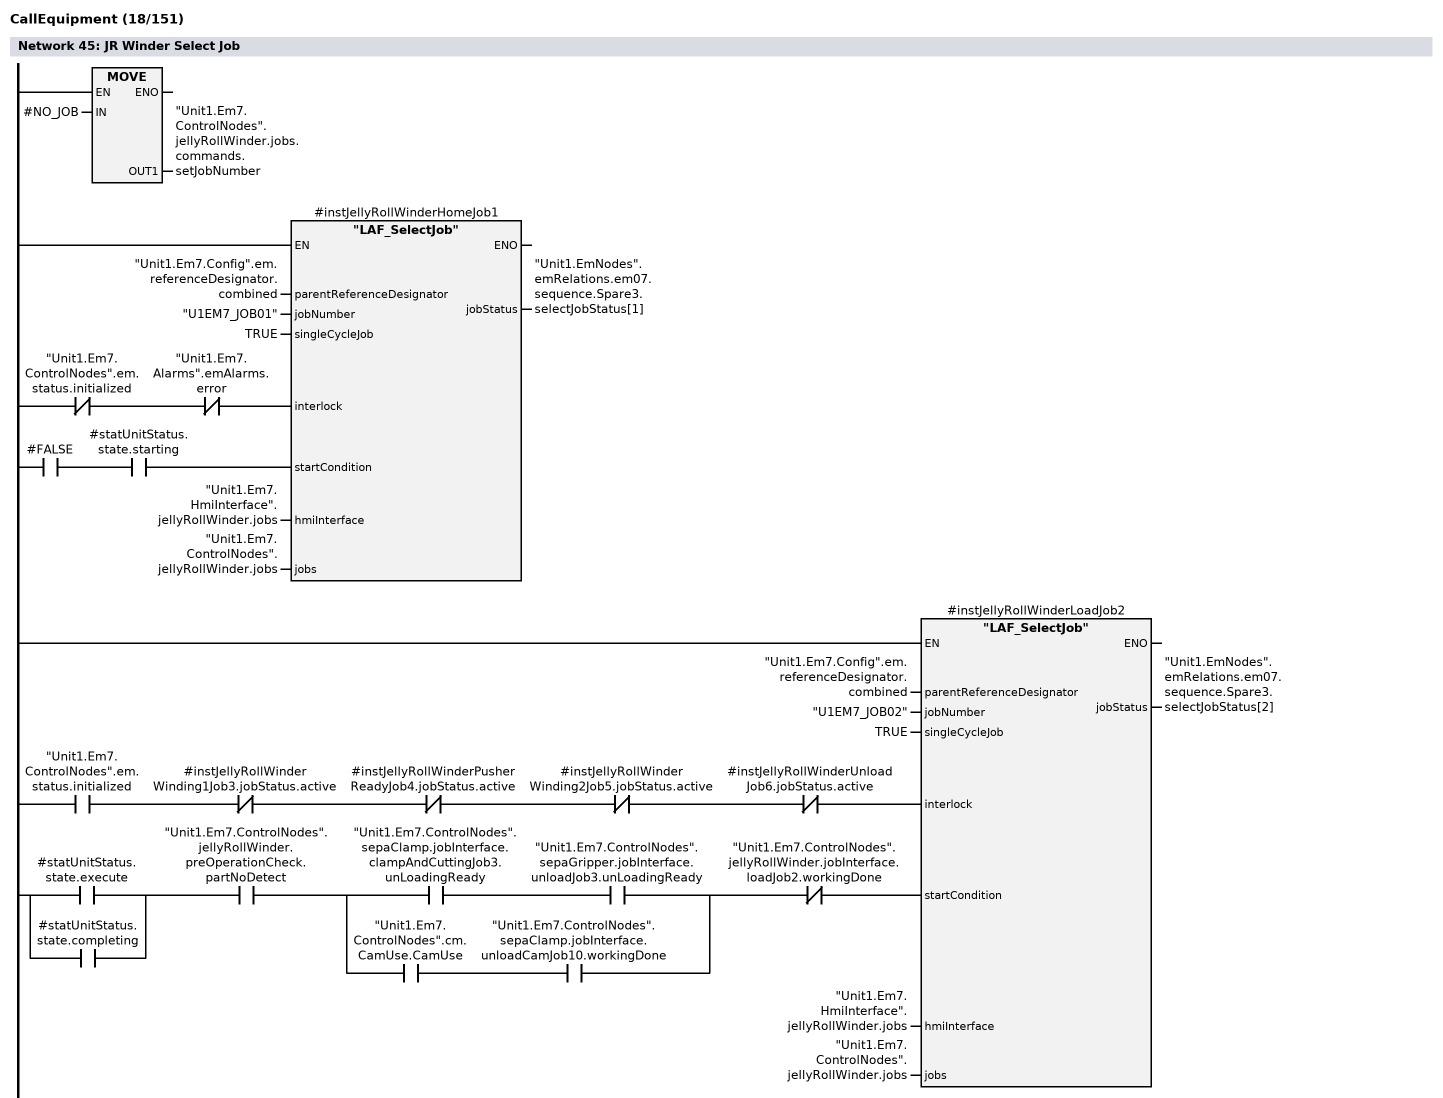
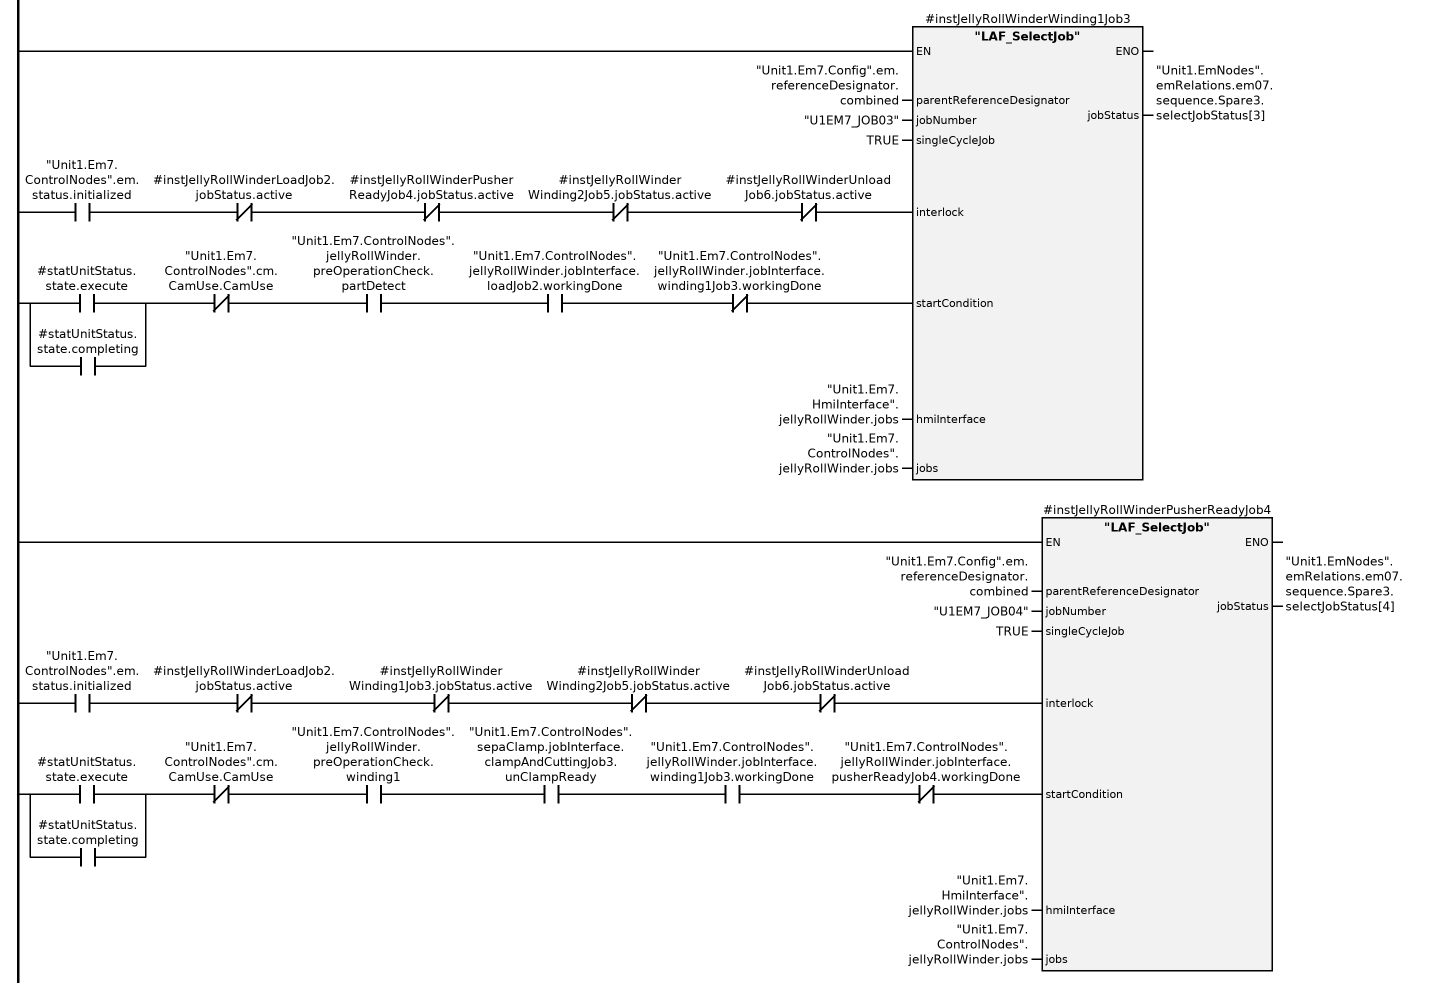
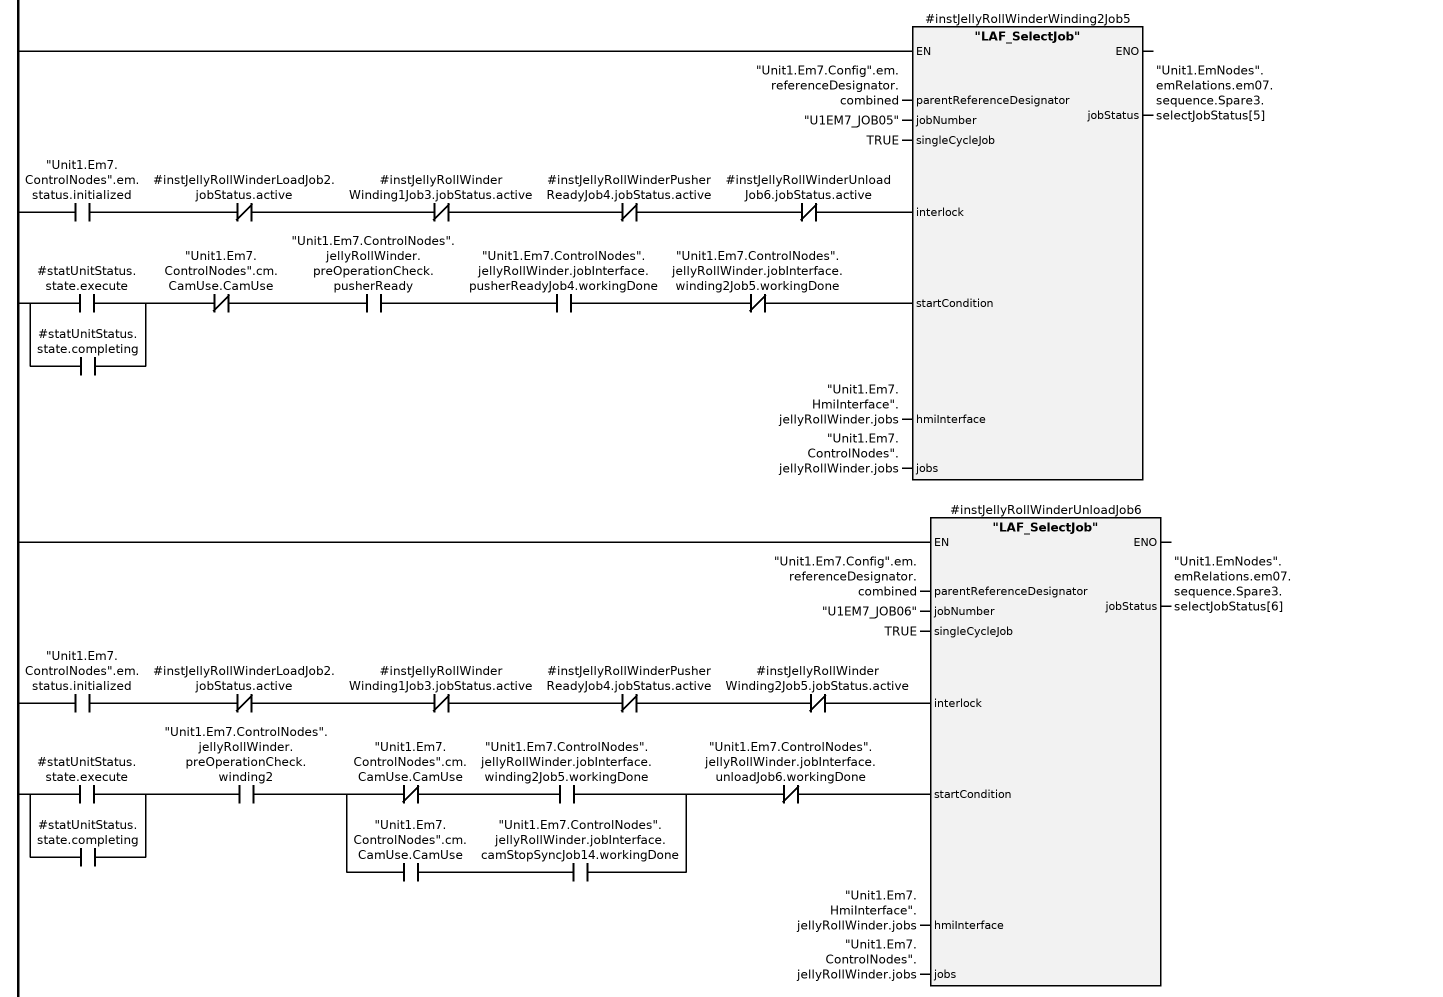
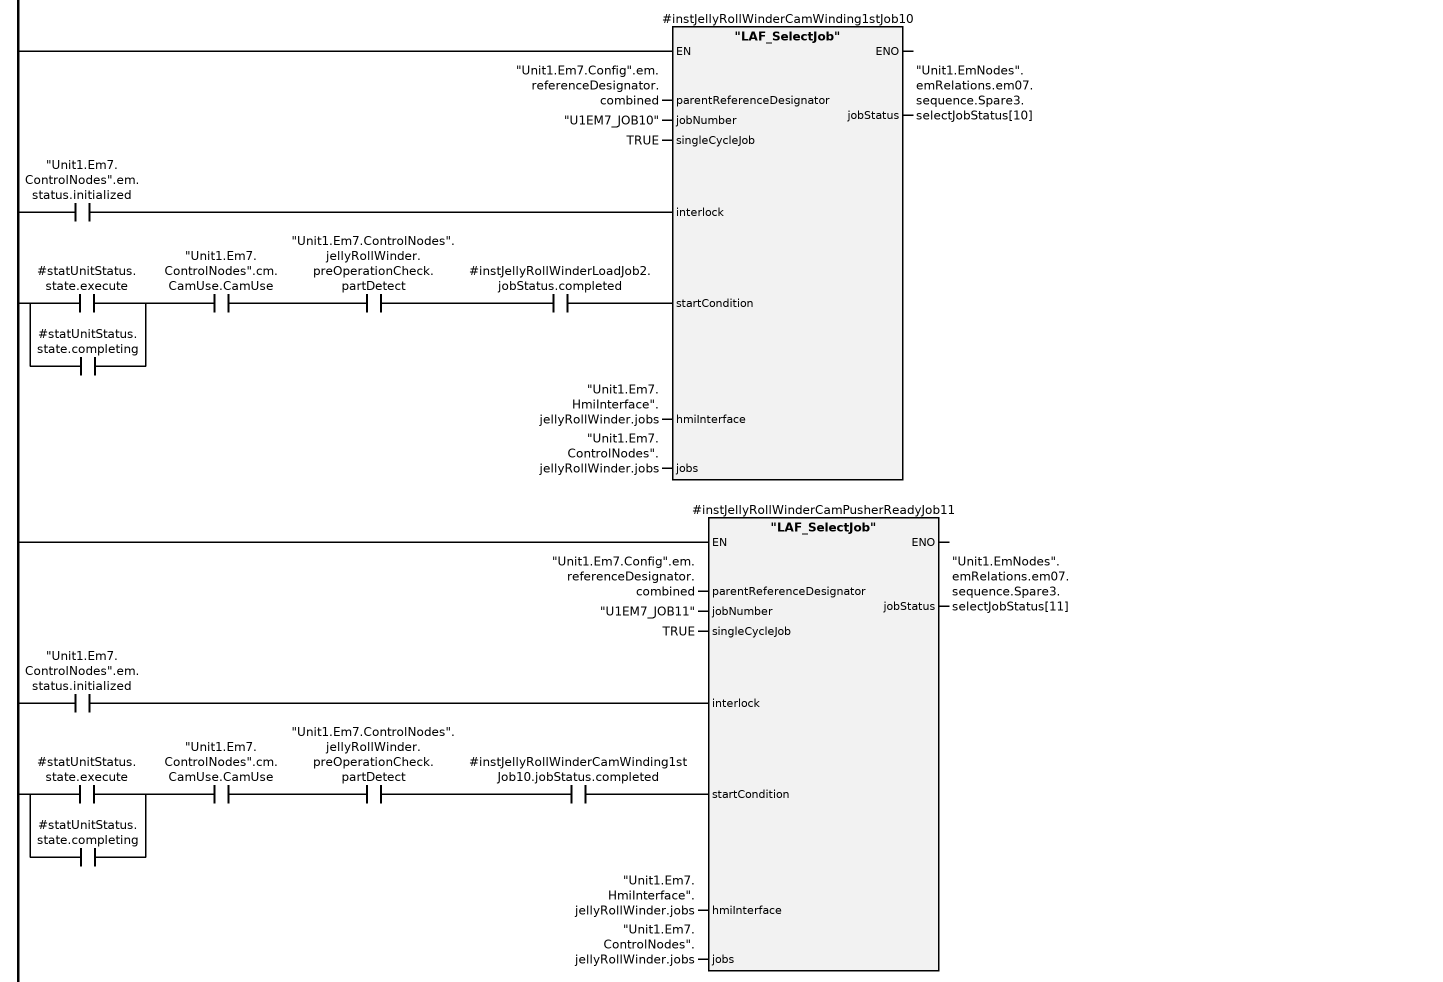
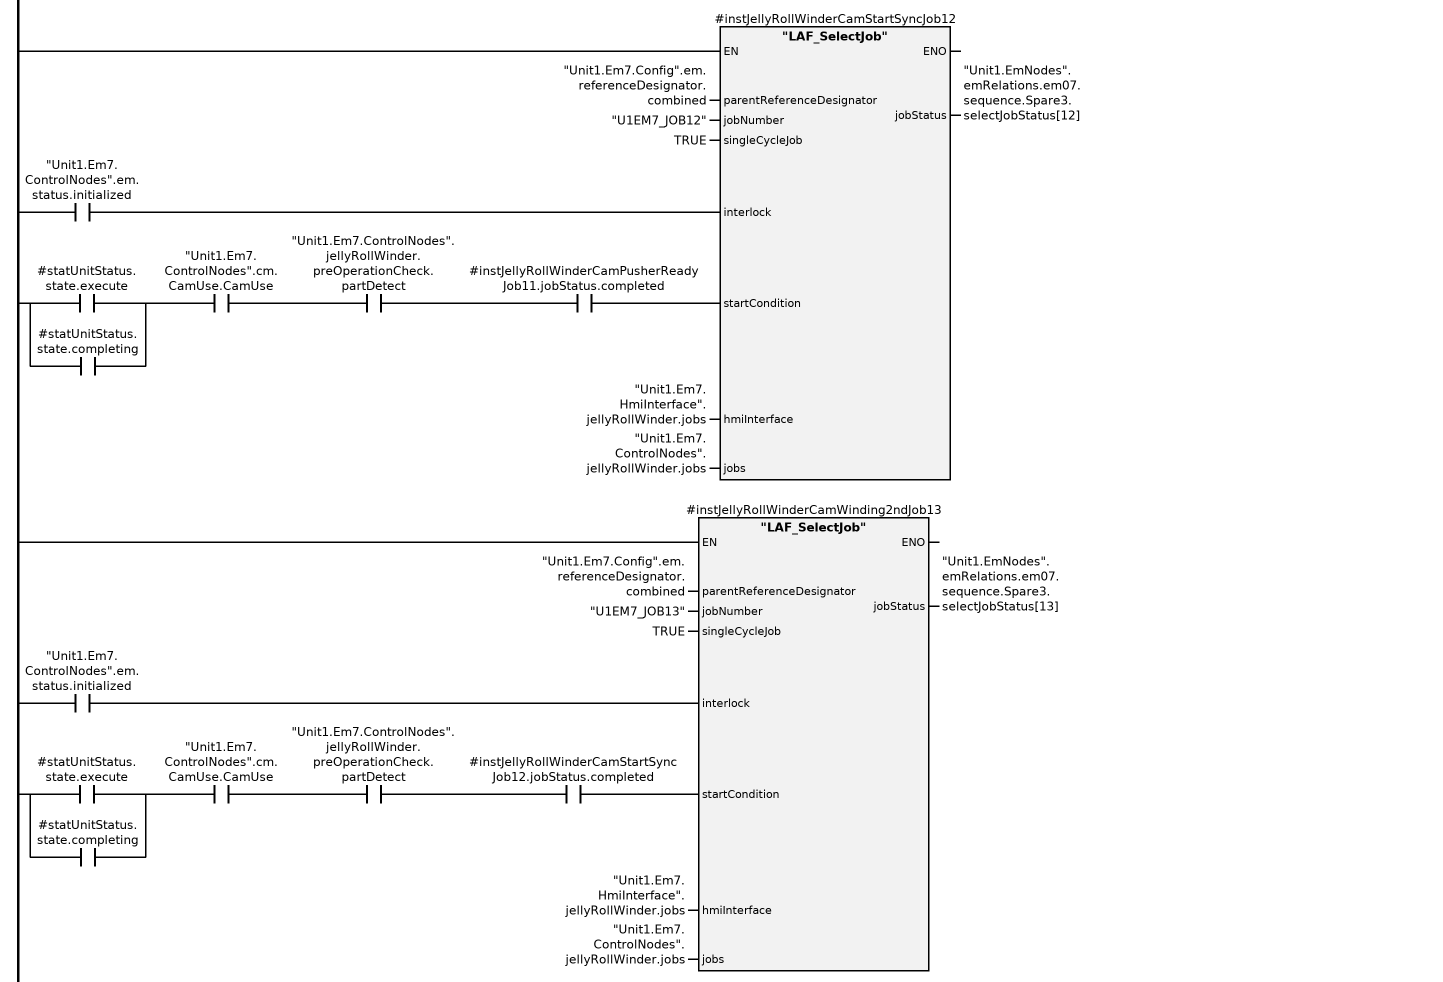
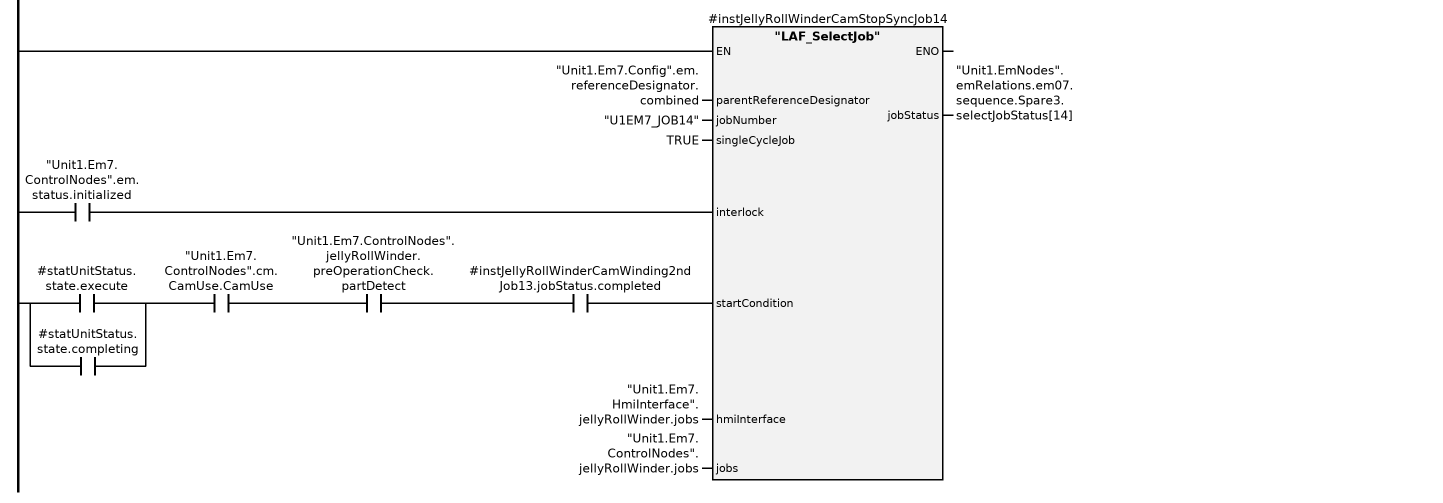
   RUNG wire#powerrail
      Move(in := #NO_JOB, out1 => "Unit1.Em7.ControlNodes".jellyRollWinder.jobs.commands.setJobNumber)
   END_RUNG
   RUNG wire#powerrail
      #instJellyRollWinderHomeJob1(interlock := wire#w1, startCondition := wire#w2, parentReferenceDesignator := "Unit1.Em7.Config".em.referenceDesignator.combined, jobNumber := "U1EM7_JOB01", singleCycleJob := TRUE, hmiInterface := "Unit1.Em7.HmiInterface".jellyRollWinder.jobs, jobs := "Unit1.Em7.ControlNodes".jellyRollWinder.jobs, jobStatus => "Unit1.EmNodes".emRelations.em07.sequence.Spare3.selectJobStatus[1])
   END_RUNG
   RUNG wire#powerrail
      I_Contact( "Unit1.Em7.ControlNodes".em.status.initialized )
      I_Contact( "Unit1.Em7.Alarms".emAlarms.error )
   END_RUNG wire#w1
   RUNG wire#powerrail
      Contact( #FALSE )
      Contact( #statUnitStatus.state.starting )
   END_RUNG wire#w2
   RUNG wire#powerrail
      #instJellyRollWinderLoadJob2(interlock := wire#w3, startCondition := wire#w7, parentReferenceDesignator := "Unit1.Em7.Config".em.referenceDesignator.combined, jobNumber := "U1EM7_JOB02", singleCycleJob := TRUE, hmiInterface := "Unit1.Em7.HmiInterface".jellyRollWinder.jobs, jobs := "Unit1.Em7.ControlNodes".jellyRollWinder.jobs, jobStatus => "Unit1.EmNodes".emRelations.em07.sequence.Spare3.selectJobStatus[2])
   END_RUNG
   RUNG wire#powerrail
      Contact( "Unit1.Em7.ControlNodes".em.status.initialized )
      I_Contact( #instJellyRollWinderWinding1Job3.jobStatus.active )
      I_Contact( #instJellyRollWinderPusherReadyJob4.jobStatus.active )
      I_Contact( #instJellyRollWinderWinding2Job5.jobStatus.active )
      I_Contact( #instJellyRollWinderUnloadJob6.jobStatus.active )
   END_RUNG wire#w3
   RUNG wire#powerrail
      Contact( #statUnitStatus.state.execute )
      wire#w4
      Contact( "Unit1.Em7.ControlNodes".jellyRollWinder.preOperationCheck.partNoDetect )
      wire#w5
      Contact( "Unit1.Em7.ControlNodes".sepaClamp.jobInterface.clampAndCuttingJob3.unLoadingReady )
      Contact( "Unit1.Em7.ControlNodes".sepaGripper.jobInterface.unloadJob3.unLoadingReady )
      wire#w6
      I_Contact( "Unit1.Em7.ControlNodes".jellyRollWinder.jobInterface.loadJob2.workingDone )
   END_RUNG wire#w7
   RUNG wire#powerrail
      Contact( #statUnitStatus.state.completing )
   END_RUNG wire#w4
   RUNG wire#w5
      Contact( "Unit1.Em7.ControlNodes".cm.CamUse.CamUse )
      Contact( "Unit1.Em7.ControlNodes".sepaClamp.jobInterface.unloadCamJob10.workingDone )
   END_RUNG wire#w6
   RUNG wire#powerrail
      #instJellyRollWinderWinding1Job3(interlock := wire#w8, startCondition := wire#w10, parentReferenceDesignator := "Unit1.Em7.Config".em.referenceDesignator.combined, jobNumber := "U1EM7_JOB03", singleCycleJob := TRUE, hmiInterface := "Unit1.Em7.HmiInterface".jellyRollWinder.jobs, jobs := "Unit1.Em7.ControlNodes".jellyRollWinder.jobs, jobStatus => "Unit1.EmNodes".emRelations.em07.sequence.Spare3.selectJobStatus[3])
   END_RUNG
   RUNG wire#powerrail
      Contact( "Unit1.Em7.ControlNodes".em.status.initialized )
      I_Contact( #instJellyRollWinderLoadJob2.jobStatus.active )
      I_Contact( #instJellyRollWinderPusherReadyJob4.jobStatus.active )
      I_Contact( #instJellyRollWinderWinding2Job5.jobStatus.active )
      I_Contact( #instJellyRollWinderUnloadJob6.jobStatus.active )
   END_RUNG wire#w8
   RUNG wire#powerrail
      Contact( #statUnitStatus.state.execute )
      wire#w9
      I_Contact( "Unit1.Em7.ControlNodes".cm.CamUse.CamUse )
      Contact( "Unit1.Em7.ControlNodes".jellyRollWinder.preOperationCheck.partDetect )
      Contact( "Unit1.Em7.ControlNodes".jellyRollWinder.jobInterface.loadJob2.workingDone )
      I_Contact( "Unit1.Em7.ControlNodes".jellyRollWinder.jobInterface.winding1Job3.workingDone )
   END_RUNG wire#w10
   RUNG wire#powerrail
      Contact( #statUnitStatus.state.completing )
   END_RUNG wire#w9
   RUNG wire#powerrail
      #instJellyRollWinderPusherReadyJob4(interlock := wire#w11, startCondition := wire#w13, parentReferenceDesignator := "Unit1.Em7.Config".em.referenceDesignator.combined, jobNumber := "U1EM7_JOB04", singleCycleJob := TRUE, hmiInterface := "Unit1.Em7.HmiInterface".jellyRollWinder.jobs, jobs := "Unit1.Em7.ControlNodes".jellyRollWinder.jobs, jobStatus => "Unit1.EmNodes".emRelations.em07.sequence.Spare3.selectJobStatus[4])
   END_RUNG
   RUNG wire#powerrail
      Contact( "Unit1.Em7.ControlNodes".em.status.initialized )
      I_Contact( #instJellyRollWinderLoadJob2.jobStatus.active )
      I_Contact( #instJellyRollWinderWinding1Job3.jobStatus.active )
      I_Contact( #instJellyRollWinderWinding2Job5.jobStatus.active )
      I_Contact( #instJellyRollWinderUnloadJob6.jobStatus.active )
   END_RUNG wire#w11
   RUNG wire#powerrail
      Contact( #statUnitStatus.state.execute )
      wire#w12
      I_Contact( "Unit1.Em7.ControlNodes".cm.CamUse.CamUse )
      Contact( "Unit1.Em7.ControlNodes".jellyRollWinder.preOperationCheck.winding1 )
      Contact( "Unit1.Em7.ControlNodes".sepaClamp.jobInterface.clampAndCuttingJob3.unClampReady )
      Contact( "Unit1.Em7.ControlNodes".jellyRollWinder.jobInterface.winding1Job3.workingDone )
      I_Contact( "Unit1.Em7.ControlNodes".jellyRollWinder.jobInterface.pusherReadyJob4.workingDone )
   END_RUNG wire#w13
   RUNG wire#powerrail
      Contact( #statUnitStatus.state.completing )
   END_RUNG wire#w12
   RUNG wire#powerrail
      #instJellyRollWinderWinding2Job5(interlock := wire#w14, startCondition := wire#w16, parentReferenceDesignator := "Unit1.Em7.Config".em.referenceDesignator.combined, jobNumber := "U1EM7_JOB05", singleCycleJob := TRUE, hmiInterface := "Unit1.Em7.HmiInterface".jellyRollWinder.jobs, jobs := "Unit1.Em7.ControlNodes".jellyRollWinder.jobs, jobStatus => "Unit1.EmNodes".emRelations.em07.sequence.Spare3.selectJobStatus[5])
   END_RUNG
   RUNG wire#powerrail
      Contact( "Unit1.Em7.ControlNodes".em.status.initialized )
      I_Contact( #instJellyRollWinderLoadJob2.jobStatus.active )
      I_Contact( #instJellyRollWinderWinding1Job3.jobStatus.active )
      I_Contact( #instJellyRollWinderPusherReadyJob4.jobStatus.active )
      I_Contact( #instJellyRollWinderUnloadJob6.jobStatus.active )
   END_RUNG wire#w14
   RUNG wire#powerrail
      Contact( #statUnitStatus.state.execute )
      wire#w15
      I_Contact( "Unit1.Em7.ControlNodes".cm.CamUse.CamUse )
      Contact( "Unit1.Em7.ControlNodes".jellyRollWinder.preOperationCheck.pusherReady )
      Contact( "Unit1.Em7.ControlNodes".jellyRollWinder.jobInterface.pusherReadyJob4.workingDone )
      I_Contact( "Unit1.Em7.ControlNodes".jellyRollWinder.jobInterface.winding2Job5.workingDone )
   END_RUNG wire#w16
   RUNG wire#powerrail
      Contact( #statUnitStatus.state.completing )
   END_RUNG wire#w15
   RUNG wire#powerrail
      #instJellyRollWinderUnloadJob6(interlock := wire#w17, startCondition := wire#w21, parentReferenceDesignator := "Unit1.Em7.Config".em.referenceDesignator.combined, jobNumber := "U1EM7_JOB06", singleCycleJob := TRUE, hmiInterface := "Unit1.Em7.HmiInterface".jellyRollWinder.jobs, jobs := "Unit1.Em7.ControlNodes".jellyRollWinder.jobs, jobStatus => "Unit1.EmNodes".emRelations.em07.sequence.Spare3.selectJobStatus[6])
   END_RUNG
   RUNG wire#powerrail
      Contact( "Unit1.Em7.ControlNodes".em.status.initialized )
      I_Contact( #instJellyRollWinderLoadJob2.jobStatus.active )
      I_Contact( #instJellyRollWinderWinding1Job3.jobStatus.active )
      I_Contact( #instJellyRollWinderPusherReadyJob4.jobStatus.active )
      I_Contact( #instJellyRollWinderWinding2Job5.jobStatus.active )
   END_RUNG wire#w17
   RUNG wire#powerrail
      Contact( #statUnitStatus.state.execute )
      wire#w18
      Contact( "Unit1.Em7.ControlNodes".jellyRollWinder.preOperationCheck.winding2 )
      wire#w19
      I_Contact( "Unit1.Em7.ControlNodes".cm.CamUse.CamUse )
      Contact( "Unit1.Em7.ControlNodes".jellyRollWinder.jobInterface.winding2Job5.workingDone )
      wire#w20
      I_Contact( "Unit1.Em7.ControlNodes".jellyRollWinder.jobInterface.unloadJob6.workingDone )
   END_RUNG wire#w21
   RUNG wire#powerrail
      Contact( #statUnitStatus.state.completing )
   END_RUNG wire#w18
   RUNG wire#w19
      Contact( "Unit1.Em7.ControlNodes".cm.CamUse.CamUse )
      Contact( "Unit1.Em7.ControlNodes".jellyRollWinder.jobInterface.camStopSyncJob14.workingDone )
   END_RUNG wire#w20
   RUNG wire#powerrail
      #instJellyRollWinderCamWinding1stJob10(interlock := wire#w22, startCondition := wire#w24, parentReferenceDesignator := "Unit1.Em7.Config".em.referenceDesignator.combined, jobNumber := "U1EM7_JOB10", singleCycleJob := TRUE, hmiInterface := "Unit1.Em7.HmiInterface".jellyRollWinder.jobs, jobs := "Unit1.Em7.ControlNodes".jellyRollWinder.jobs, jobStatus => "Unit1.EmNodes".emRelations.em07.sequence.Spare3.selectJobStatus[10])
   END_RUNG
   RUNG wire#powerrail
      Contact( "Unit1.Em7.ControlNodes".em.status.initialized )
   END_RUNG wire#w22
   RUNG wire#powerrail
      Contact( #statUnitStatus.state.execute )
      wire#w23
      Contact( "Unit1.Em7.ControlNodes".cm.CamUse.CamUse )
      Contact( "Unit1.Em7.ControlNodes".jellyRollWinder.preOperationCheck.partDetect )
      Contact( #instJellyRollWinderLoadJob2.jobStatus.completed )
   END_RUNG wire#w24
   RUNG wire#powerrail
      Contact( #statUnitStatus.state.completing )
   END_RUNG wire#w23
   RUNG wire#powerrail
      #instJellyRollWinderCamPusherReadyJob11(interlock := wire#w25, startCondition := wire#w27, parentReferenceDesignator := "Unit1.Em7.Config".em.referenceDesignator.combined, jobNumber := "U1EM7_JOB11", singleCycleJob := TRUE, hmiInterface := "Unit1.Em7.HmiInterface".jellyRollWinder.jobs, jobs := "Unit1.Em7.ControlNodes".jellyRollWinder.jobs, jobStatus => "Unit1.EmNodes".emRelations.em07.sequence.Spare3.selectJobStatus[11])
   END_RUNG
   RUNG wire#powerrail
      Contact( "Unit1.Em7.ControlNodes".em.status.initialized )
   END_RUNG wire#w25
   RUNG wire#powerrail
      Contact( #statUnitStatus.state.execute )
      wire#w26
      Contact( "Unit1.Em7.ControlNodes".cm.CamUse.CamUse )
      Contact( "Unit1.Em7.ControlNodes".jellyRollWinder.preOperationCheck.partDetect )
      Contact( #instJellyRollWinderCamWinding1stJob10.jobStatus.completed )
   END_RUNG wire#w27
   RUNG wire#powerrail
      Contact( #statUnitStatus.state.completing )
   END_RUNG wire#w26
   RUNG wire#powerrail
      #instJellyRollWinderCamStartSyncJob12(interlock := wire#w28, startCondition := wire#w30, parentReferenceDesignator := "Unit1.Em7.Config".em.referenceDesignator.combined, jobNumber := "U1EM7_JOB12", singleCycleJob := TRUE, hmiInterface := "Unit1.Em7.HmiInterface".jellyRollWinder.jobs, jobs := "Unit1.Em7.ControlNodes".jellyRollWinder.jobs, jobStatus => "Unit1.EmNodes".emRelations.em07.sequence.Spare3.selectJobStatus[12])
   END_RUNG
   RUNG wire#powerrail
      Contact( "Unit1.Em7.ControlNodes".em.status.initialized )
   END_RUNG wire#w28
   RUNG wire#powerrail
      Contact( #statUnitStatus.state.execute )
      wire#w29
      Contact( "Unit1.Em7.ControlNodes".cm.CamUse.CamUse )
      Contact( "Unit1.Em7.ControlNodes".jellyRollWinder.preOperationCheck.partDetect )
      Contact( #instJellyRollWinderCamPusherReadyJob11.jobStatus.completed )
   END_RUNG wire#w30
   RUNG wire#powerrail
      Contact( #statUnitStatus.state.completing )
   END_RUNG wire#w29
   RUNG wire#powerrail
      #instJellyRollWinderCamWinding2ndJob13(interlock := wire#w31, startCondition := wire#w33, parentReferenceDesignator := "Unit1.Em7.Config".em.referenceDesignator.combined, jobNumber := "U1EM7_JOB13", singleCycleJob := TRUE, hmiInterface := "Unit1.Em7.HmiInterface".jellyRollWinder.jobs, jobs := "Unit1.Em7.ControlNodes".jellyRollWinder.jobs, jobStatus => "Unit1.EmNodes".emRelations.em07.sequence.Spare3.selectJobStatus[13])
   END_RUNG
   RUNG wire#powerrail
      Contact( "Unit1.Em7.ControlNodes".em.status.initialized )
   END_RUNG wire#w31
   RUNG wire#powerrail
      Contact( #statUnitStatus.state.execute )
      wire#w32
      Contact( "Unit1.Em7.ControlNodes".cm.CamUse.CamUse )
      Contact( "Unit1.Em7.ControlNodes".jellyRollWinder.preOperationCheck.partDetect )
      Contact( #instJellyRollWinderCamStartSyncJob12.jobStatus.completed )
   END_RUNG wire#w33
   RUNG wire#powerrail
      Contact( #statUnitStatus.state.completing )
   END_RUNG wire#w32
   RUNG wire#powerrail
      #instJellyRollWinderCamStopSyncJob14(interlock := wire#w34, startCondition := wire#w36, parentReferenceDesignator := "Unit1.Em7.Config".em.referenceDesignator.combined, jobNumber := "U1EM7_JOB14", singleCycleJob := TRUE, hmiInterface := "Unit1.Em7.HmiInterface".jellyRollWinder.jobs, jobs := "Unit1.Em7.ControlNodes".jellyRollWinder.jobs, jobStatus => "Unit1.EmNodes".emRelations.em07.sequence.Spare3.selectJobStatus[14])
   END_RUNG
   RUNG wire#powerrail
      Contact( "Unit1.Em7.ControlNodes".em.status.initialized )
   END_RUNG wire#w34
   RUNG wire#powerrail
      Contact( #statUnitStatus.state.execute )
      wire#w35
      Contact( "Unit1.Em7.ControlNodes".cm.CamUse.CamUse )
      Contact( "Unit1.Em7.ControlNodes".jellyRollWinder.preOperationCheck.partDetect )
      Contact( #instJellyRollWinderCamWinding2ndJob13.jobStatus.completed )
   END_RUNG wire#w36
   RUNG wire#powerrail
      Contact( #statUnitStatus.state.completing )
   END_RUNG wire#w35
   // the same network as SCL:
   "Unit1.Em7.ControlNodes".jellyRollWinder.jobs.commands.setJobNumber := #NO_JOB;
   #instJellyRollWinderHomeJob1(parentReferenceDesignator := "Unit1.Em7.Config".em.referenceDesignator.combined,   // "LAF_SelectJob"
                           jobNumber := "U1EM7_JOB01",
                           singleCycleJob := TRUE,
                           interlock := NOT "Unit1.Em7.ControlNodes".em.status.initialized AND NOT "Unit1.Em7.Alarms".emAlarms.error,
                           startCondition := #FALSE AND #statUnitStatus.state.starting,
                           hmiInterface := "Unit1.Em7.HmiInterface".jellyRollWinder.jobs,
                           jobs := "Unit1.Em7.ControlNodes".jellyRollWinder.jobs,
                           jobStatus => "Unit1.EmNodes".emRelations.em07.sequence.Spare3.selectJobStatus[1]);
   #instJellyRollWinderLoadJob2(parentReferenceDesignator := "Unit1.Em7.Config".em.referenceDesignator.combined,   // "LAF_SelectJob"
                           jobNumber := "U1EM7_JOB02",
                           singleCycleJob := TRUE,
                           interlock := "Unit1.Em7.ControlNodes".em.status.initialized AND NOT #instJellyRollWinderWinding1Job3.jobStatus.active AND NOT #instJellyRollWinderPusherReadyJob4.jobStatus.active AND NOT #instJellyRollWinderWinding2Job5.jobStatus.active AND NOT #instJellyRollWinderUnloadJob6.jobStatus.active,
                           startCondition := (#statUnitStatus.state.execute OR #statUnitStatus.state.completing) AND "Unit1.Em7.ControlNodes".jellyRollWinder.preOperationCheck.partNoDetect AND (("Unit1.Em7.ControlNodes".sepaClamp.jobInterface.clampAndCuttingJob3.unLoadingReady AND "Unit1.Em7.ControlNodes".sepaGripper.jobInterface.unloadJob3.unLoadingReady) OR ("Unit1.Em7.ControlNodes".cm.CamUse.CamUse AND "Unit1.Em7.ControlNodes".sepaClamp.jobInterface.unloadCamJob10.workingDone)) AND NOT "Unit1.Em7.ControlNodes".jellyRollWinder.jobInterface.loadJob2.workingDone,
                           hmiInterface := "Unit1.Em7.HmiInterface".jellyRollWinder.jobs,
                           jobs := "Unit1.Em7.ControlNodes".jellyRollWinder.jobs,
                           jobStatus => "Unit1.EmNodes".emRelations.em07.sequence.Spare3.selectJobStatus[2]);
   #instJellyRollWinderWinding1Job3(parentReferenceDesignator := "Unit1.Em7.Config".em.referenceDesignator.combined,   // "LAF_SelectJob"
                           jobNumber := "U1EM7_JOB03",
                           singleCycleJob := TRUE,
                           interlock := "Unit1.Em7.ControlNodes".em.status.initialized AND NOT #instJellyRollWinderLoadJob2.jobStatus.active AND NOT #instJellyRollWinderPusherReadyJob4.jobStatus.active AND NOT #instJellyRollWinderWinding2Job5.jobStatus.active AND NOT #instJellyRollWinderUnloadJob6.jobStatus.active,
                           startCondition := (#statUnitStatus.state.execute OR #statUnitStatus.state.completing) AND NOT "Unit1.Em7.ControlNodes".cm.CamUse.CamUse AND "Unit1.Em7.ControlNodes".jellyRollWinder.preOperationCheck.partDetect AND "Unit1.Em7.ControlNodes".jellyRollWinder.jobInterface.loadJob2.workingDone AND NOT "Unit1.Em7.ControlNodes".jellyRollWinder.jobInterface.winding1Job3.workingDone,
                           hmiInterface := "Unit1.Em7.HmiInterface".jellyRollWinder.jobs,
                           jobs := "Unit1.Em7.ControlNodes".jellyRollWinder.jobs,
                           jobStatus => "Unit1.EmNodes".emRelations.em07.sequence.Spare3.selectJobStatus[3]);
   #instJellyRollWinderPusherReadyJob4(parentReferenceDesignator := "Unit1.Em7.Config".em.referenceDesignator.combined,   // "LAF_SelectJob"
                           jobNumber := "U1EM7_JOB04",
                           singleCycleJob := TRUE,
                           interlock := "Unit1.Em7.ControlNodes".em.status.initialized AND NOT #instJellyRollWinderLoadJob2.jobStatus.active AND NOT #instJellyRollWinderWinding1Job3.jobStatus.active AND NOT #instJellyRollWinderWinding2Job5.jobStatus.active AND NOT #instJellyRollWinderUnloadJob6.jobStatus.active,
                           startCondition := (#statUnitStatus.state.execute OR #statUnitStatus.state.completing) AND NOT "Unit1.Em7.ControlNodes".cm.CamUse.CamUse AND "Unit1.Em7.ControlNodes".jellyRollWinder.preOperationCheck.winding1 AND "Unit1.Em7.ControlNodes".sepaClamp.jobInterface.clampAndCuttingJob3.unClampReady AND "Unit1.Em7.ControlNodes".jellyRollWinder.jobInterface.winding1Job3.workingDone AND NOT "Unit1.Em7.ControlNodes".jellyRollWinder.jobInterface.pusherReadyJob4.workingDone,
                           hmiInterface := "Unit1.Em7.HmiInterface".jellyRollWinder.jobs,
                           jobs := "Unit1.Em7.ControlNodes".jellyRollWinder.jobs,
                           jobStatus => "Unit1.EmNodes".emRelations.em07.sequence.Spare3.selectJobStatus[4]);
   #instJellyRollWinderWinding2Job5(parentReferenceDesignator := "Unit1.Em7.Config".em.referenceDesignator.combined,   // "LAF_SelectJob"
                           jobNumber := "U1EM7_JOB05",
                           singleCycleJob := TRUE,
                           interlock := "Unit1.Em7.ControlNodes".em.status.initialized AND NOT #instJellyRollWinderLoadJob2.jobStatus.active AND NOT #instJellyRollWinderWinding1Job3.jobStatus.active AND NOT #instJellyRollWinderPusherReadyJob4.jobStatus.active AND NOT #instJellyRollWinderUnloadJob6.jobStatus.active,
                           startCondition := (#statUnitStatus.state.execute OR #statUnitStatus.state.completing) AND NOT "Unit1.Em7.ControlNodes".cm.CamUse.CamUse AND "Unit1.Em7.ControlNodes".jellyRollWinder.preOperationCheck.pusherReady AND "Unit1.Em7.ControlNodes".jellyRollWinder.jobInterface.pusherReadyJob4.workingDone AND NOT "Unit1.Em7.ControlNodes".jellyRollWinder.jobInterface.winding2Job5.workingDone,
                           hmiInterface := "Unit1.Em7.HmiInterface".jellyRollWinder.jobs,
                           jobs := "Unit1.Em7.ControlNodes".jellyRollWinder.jobs,
                           jobStatus => "Unit1.EmNodes".emRelations.em07.sequence.Spare3.selectJobStatus[5]);
   #instJellyRollWinderUnloadJob6(parentReferenceDesignator := "Unit1.Em7.Config".em.referenceDesignator.combined,   // "LAF_SelectJob"
                           jobNumber := "U1EM7_JOB06",
                           singleCycleJob := TRUE,
                           interlock := "Unit1.Em7.ControlNodes".em.status.initialized AND NOT #instJellyRollWinderLoadJob2.jobStatus.active AND NOT #instJellyRollWinderWinding1Job3.jobStatus.active AND NOT #instJellyRollWinderPusherReadyJob4.jobStatus.active AND NOT #instJellyRollWinderWinding2Job5.jobStatus.active,
                           startCondition := (#statUnitStatus.state.execute OR #statUnitStatus.state.completing) AND "Unit1.Em7.ControlNodes".jellyRollWinder.preOperationCheck.winding2 AND ((NOT "Unit1.Em7.ControlNodes".cm.CamUse.CamUse AND "Unit1.Em7.ControlNodes".jellyRollWinder.jobInterface.winding2Job5.workingDone) OR ("Unit1.Em7.ControlNodes".cm.CamUse.CamUse AND "Unit1.Em7.ControlNodes".jellyRollWinder.jobInterface.camStopSyncJob14.workingDone)) AND NOT "Unit1.Em7.ControlNodes".jellyRollWinder.jobInterface.unloadJob6.workingDone,
                           hmiInterface := "Unit1.Em7.HmiInterface".jellyRollWinder.jobs,
                           jobs := "Unit1.Em7.ControlNodes".jellyRollWinder.jobs,
                           jobStatus => "Unit1.EmNodes".emRelations.em07.sequence.Spare3.selectJobStatus[6]);
   #instJellyRollWinderCamWinding1stJob10(parentReferenceDesignator := "Unit1.Em7.Config".em.referenceDesignator.combined,   // "LAF_SelectJob"
                           jobNumber := "U1EM7_JOB10",
                           singleCycleJob := TRUE,
                           interlock := "Unit1.Em7.ControlNodes".em.status.initialized,
                           startCondition := (#statUnitStatus.state.execute OR #statUnitStatus.state.completing) AND "Unit1.Em7.ControlNodes".cm.CamUse.CamUse AND "Unit1.Em7.ControlNodes".jellyRollWinder.preOperationCheck.partDetect AND #instJellyRollWinderLoadJob2.jobStatus.completed,
                           hmiInterface := "Unit1.Em7.HmiInterface".jellyRollWinder.jobs,
                           jobs := "Unit1.Em7.ControlNodes".jellyRollWinder.jobs,
                           jobStatus => "Unit1.EmNodes".emRelations.em07.sequence.Spare3.selectJobStatus[10]);
   #instJellyRollWinderCamPusherReadyJob11(parentReferenceDesignator := "Unit1.Em7.Config".em.referenceDesignator.combined,   // "LAF_SelectJob"
                           jobNumber := "U1EM7_JOB11",
                           singleCycleJob := TRUE,
                           interlock := "Unit1.Em7.ControlNodes".em.status.initialized,
                           startCondition := (#statUnitStatus.state.execute OR #statUnitStatus.state.completing) AND "Unit1.Em7.ControlNodes".cm.CamUse.CamUse AND "Unit1.Em7.ControlNodes".jellyRollWinder.preOperationCheck.partDetect AND #instJellyRollWinderCamWinding1stJob10.jobStatus.completed,
                           hmiInterface := "Unit1.Em7.HmiInterface".jellyRollWinder.jobs,
                           jobs := "Unit1.Em7.ControlNodes".jellyRollWinder.jobs,
                           jobStatus => "Unit1.EmNodes".emRelations.em07.sequence.Spare3.selectJobStatus[11]);
   #instJellyRollWinderCamStartSyncJob12(parentReferenceDesignator := "Unit1.Em7.Config".em.referenceDesignator.combined,   // "LAF_SelectJob"
                           jobNumber := "U1EM7_JOB12",
                           singleCycleJob := TRUE,
                           interlock := "Unit1.Em7.ControlNodes".em.status.initialized,
                           startCondition := (#statUnitStatus.state.execute OR #statUnitStatus.state.completing) AND "Unit1.Em7.ControlNodes".cm.CamUse.CamUse AND "Unit1.Em7.ControlNodes".jellyRollWinder.preOperationCheck.partDetect AND #instJellyRollWinderCamPusherReadyJob11.jobStatus.completed,
                           hmiInterface := "Unit1.Em7.HmiInterface".jellyRollWinder.jobs,
                           jobs := "Unit1.Em7.ControlNodes".jellyRollWinder.jobs,
                           jobStatus => "Unit1.EmNodes".emRelations.em07.sequence.Spare3.selectJobStatus[12]);
   #instJellyRollWinderCamWinding2ndJob13(parentReferenceDesignator := "Unit1.Em7.Config".em.referenceDesignator.combined,   // "LAF_SelectJob"
                           jobNumber := "U1EM7_JOB13",
                           singleCycleJob := TRUE,
                           interlock := "Unit1.Em7.ControlNodes".em.status.initialized,
                           startCondition := (#statUnitStatus.state.execute OR #statUnitStatus.state.completing) AND "Unit1.Em7.ControlNodes".cm.CamUse.CamUse AND "Unit1.Em7.ControlNodes".jellyRollWinder.preOperationCheck.partDetect AND #instJellyRollWinderCamStartSyncJob12.jobStatus.completed,
                           hmiInterface := "Unit1.Em7.HmiInterface".jellyRollWinder.jobs,
                           jobs := "Unit1.Em7.ControlNodes".jellyRollWinder.jobs,
                           jobStatus => "Unit1.EmNodes".emRelations.em07.sequence.Spare3.selectJobStatus[13]);
   #instJellyRollWinderCamStopSyncJob14(parentReferenceDesignator := "Unit1.Em7.Config".em.referenceDesignator.combined,   // "LAF_SelectJob"
                           jobNumber := "U1EM7_JOB14",
                           singleCycleJob := TRUE,
                           interlock := "Unit1.Em7.ControlNodes".em.status.initialized,
                           startCondition := (#statUnitStatus.state.execute OR #statUnitStatus.state.completing) AND "Unit1.Em7.ControlNodes".cm.CamUse.CamUse AND "Unit1.Em7.ControlNodes".jellyRollWinder.preOperationCheck.partDetect AND #instJellyRollWinderCamWinding2ndJob13.jobStatus.completed,
                           hmiInterface := "Unit1.Em7.HmiInterface".jellyRollWinder.jobs,
                           jobs := "Unit1.Em7.ControlNodes".jellyRollWinder.jobs,
                           jobStatus => "Unit1.EmNodes".emRelations.em07.sequence.Spare3.selectJobStatus[14]);
END_REGION

REGION Network 46: JR Winder Job Interface [Loading]
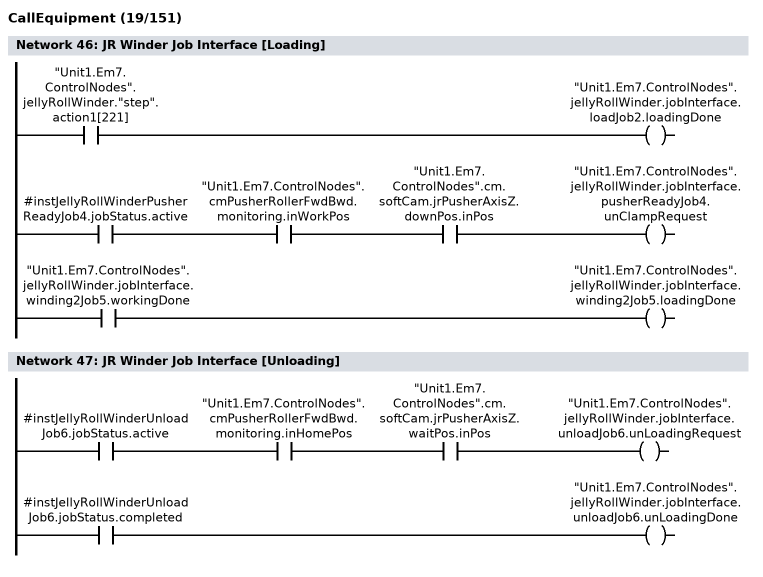
   RUNG wire#powerrail
      Contact( "Unit1.Em7.ControlNodes".jellyRollWinder."step".action1[221] )
      Coil( "Unit1.Em7.ControlNodes".jellyRollWinder.jobInterface.loadJob2.loadingDone )
   END_RUNG
   RUNG wire#powerrail
      Contact( #instJellyRollWinderPusherReadyJob4.jobStatus.active )
      Contact( "Unit1.Em7.ControlNodes".cmPusherRollerFwdBwd.monitoring.inWorkPos )
      Contact( "Unit1.Em7.ControlNodes".cm.softCam.jrPusherAxisZ.downPos.inPos )
      Coil( "Unit1.Em7.ControlNodes".jellyRollWinder.jobInterface.pusherReadyJob4.unClampRequest )
   END_RUNG
   RUNG wire#powerrail
      Contact( "Unit1.Em7.ControlNodes".jellyRollWinder.jobInterface.winding2Job5.workingDone )
      Coil( "Unit1.Em7.ControlNodes".jellyRollWinder.jobInterface.winding2Job5.loadingDone )
   END_RUNG
   // the same network as SCL:
   "Unit1.Em7.ControlNodes".jellyRollWinder.jobInterface.loadJob2.loadingDone := "Unit1.Em7.ControlNodes".jellyRollWinder."step".action1[221];
   "Unit1.Em7.ControlNodes".jellyRollWinder.jobInterface.pusherReadyJob4.unClampRequest := #instJellyRollWinderPusherReadyJob4.jobStatus.active AND "Unit1.Em7.ControlNodes".cmPusherRollerFwdBwd.monitoring.inWorkPos AND "Unit1.Em7.ControlNodes".cm.softCam.jrPusherAxisZ.downPos.inPos;
   "Unit1.Em7.ControlNodes".jellyRollWinder.jobInterface.winding2Job5.loadingDone := "Unit1.Em7.ControlNodes".jellyRollWinder.jobInterface.winding2Job5.workingDone;
END_REGION

REGION Network 47: JR Winder Job Interface [Unloading]
   RUNG wire#powerrail
      Contact( #instJellyRollWinderUnloadJob6.jobStatus.active )
      Contact( "Unit1.Em7.ControlNodes".cmPusherRollerFwdBwd.monitoring.inHomePos )
      Contact( "Unit1.Em7.ControlNodes".cm.softCam.jrPusherAxisZ.waitPos.inPos )
      Coil( "Unit1.Em7.ControlNodes".jellyRollWinder.jobInterface.unloadJob6.unLoadingRequest )
   END_RUNG
   RUNG wire#powerrail
      Contact( #instJellyRollWinderUnloadJob6.jobStatus.completed )
      Coil( "Unit1.Em7.ControlNodes".jellyRollWinder.jobInterface.unloadJob6.unLoadingDone )
   END_RUNG
   // the same network as SCL:
   "Unit1.Em7.ControlNodes".jellyRollWinder.jobInterface.unloadJob6.unLoadingRequest := #instJellyRollWinderUnloadJob6.jobStatus.active AND "Unit1.Em7.ControlNodes".cmPusherRollerFwdBwd.monitoring.inHomePos AND "Unit1.Em7.ControlNodes".cm.softCam.jrPusherAxisZ.waitPos.inPos;
   "Unit1.Em7.ControlNodes".jellyRollWinder.jobInterface.unloadJob6.unLoadingDone := #instJellyRollWinderUnloadJob6.jobStatus.completed;
END_REGION

REGION Network 48: JR Winder Job Interface Working Done
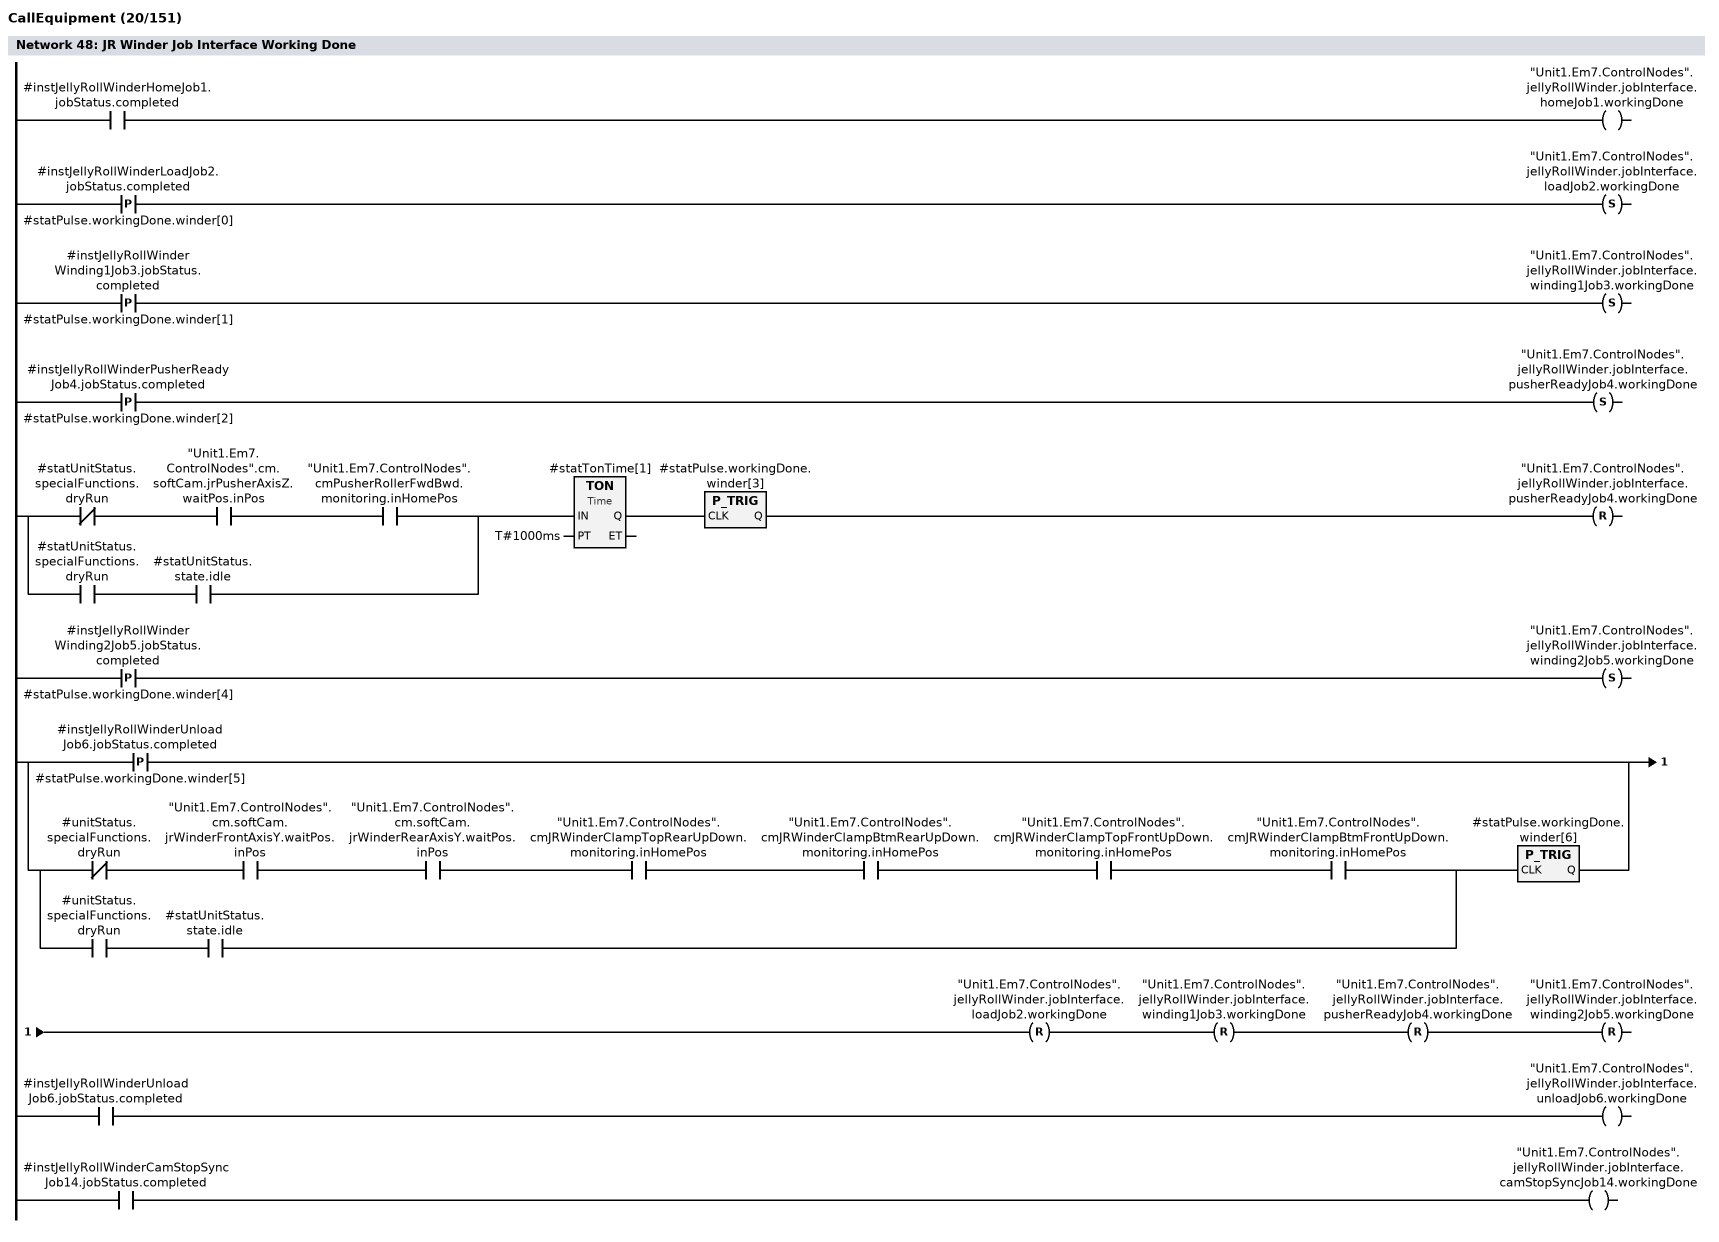
   RUNG wire#powerrail
      Contact( #instJellyRollWinderHomeJob1.jobStatus.completed )
      Coil( "Unit1.Em7.ControlNodes".jellyRollWinder.jobInterface.homeJob1.workingDone )
   END_RUNG
   RUNG wire#powerrail
      P_Contact(operand := #instJellyRollWinderLoadJob2.jobStatus.completed, bit := #statPulse.workingDone.winder[0])
      S_Coil( "Unit1.Em7.ControlNodes".jellyRollWinder.jobInterface.loadJob2.workingDone )
   END_RUNG
   RUNG wire#powerrail
      P_Contact(operand := #instJellyRollWinderWinding1Job3.jobStatus.completed, bit := #statPulse.workingDone.winder[1])
      S_Coil( "Unit1.Em7.ControlNodes".jellyRollWinder.jobInterface.winding1Job3.workingDone )
   END_RUNG
   RUNG wire#powerrail
      P_Contact(operand := #instJellyRollWinderPusherReadyJob4.jobStatus.completed, bit := #statPulse.workingDone.winder[2])
      S_Coil( "Unit1.Em7.ControlNodes".jellyRollWinder.jobInterface.pusherReadyJob4.workingDone )
   END_RUNG
   RUNG wire#powerrail
      I_Contact( #statUnitStatus.specialFunctions.dryRun )
      Contact( "Unit1.Em7.ControlNodes".cm.softCam.jrPusherAxisZ.waitPos.inPos )
      Contact( "Unit1.Em7.ControlNodes".cmPusherRollerFwdBwd.monitoring.inHomePos )
      wire#w1
      { S7_Templates := "time_type := Time" } #statTonTime[1].TON(pt := T#1000ms, et =>)
      P_Trig( #statPulse.workingDone.winder[3] )
      R_Coil( "Unit1.Em7.ControlNodes".jellyRollWinder.jobInterface.pusherReadyJob4.workingDone )
   END_RUNG
   RUNG wire#powerrail
      Contact( #statUnitStatus.specialFunctions.dryRun )
      Contact( #statUnitStatus.state.idle )
   END_RUNG wire#w1
   RUNG wire#powerrail
      P_Contact(operand := #instJellyRollWinderWinding2Job5.jobStatus.completed, bit := #statPulse.workingDone.winder[4])
      S_Coil( "Unit1.Em7.ControlNodes".jellyRollWinder.jobInterface.winding2Job5.workingDone )
   END_RUNG
   RUNG wire#powerrail
      P_Contact(operand := #instJellyRollWinderUnloadJob6.jobStatus.completed, bit := #statPulse.workingDone.winder[5])
      wire#w2
      R_Coil( "Unit1.Em7.ControlNodes".jellyRollWinder.jobInterface.loadJob2.workingDone )
      R_Coil( "Unit1.Em7.ControlNodes".jellyRollWinder.jobInterface.winding1Job3.workingDone )
      R_Coil( "Unit1.Em7.ControlNodes".jellyRollWinder.jobInterface.pusherReadyJob4.workingDone )
      R_Coil( "Unit1.Em7.ControlNodes".jellyRollWinder.jobInterface.winding2Job5.workingDone )
   END_RUNG
   RUNG wire#powerrail
      I_Contact( #unitStatus.specialFunctions.dryRun )
      Contact( "Unit1.Em7.ControlNodes".cm.softCam.jrWinderFrontAxisY.waitPos.inPos )
      Contact( "Unit1.Em7.ControlNodes".cm.softCam.jrWinderRearAxisY.waitPos.inPos )
      Contact( "Unit1.Em7.ControlNodes".cmJRWinderClampTopRearUpDown.monitoring.inHomePos )
      Contact( "Unit1.Em7.ControlNodes".cmJRWinderClampBtmRearUpDown.monitoring.inHomePos )
      Contact( "Unit1.Em7.ControlNodes".cmJRWinderClampTopFrontUpDown.monitoring.inHomePos )
      Contact( "Unit1.Em7.ControlNodes".cmJRWinderClampBtmFrontUpDown.monitoring.inHomePos )
      wire#w3
      P_Trig( #statPulse.workingDone.winder[6] )
   END_RUNG wire#w2
   RUNG wire#powerrail
      Contact( #unitStatus.specialFunctions.dryRun )
      Contact( #statUnitStatus.state.idle )
   END_RUNG wire#w3
   RUNG wire#powerrail
      Contact( #instJellyRollWinderUnloadJob6.jobStatus.completed )
      Coil( "Unit1.Em7.ControlNodes".jellyRollWinder.jobInterface.unloadJob6.workingDone )
   END_RUNG
   RUNG wire#powerrail
      Contact( #instJellyRollWinderCamStopSyncJob14.jobStatus.completed )
      Coil( "Unit1.Em7.ControlNodes".jellyRollWinder.jobInterface.camStopSyncJob14.workingDone )
   END_RUNG
   // the same network as SCL:
   "Unit1.Em7.ControlNodes".jellyRollWinder.jobInterface.homeJob1.workingDone := #instJellyRollWinderHomeJob1.jobStatus.completed;
   #_w1 := #instJellyRollWinderLoadJob2.jobStatus.completed AND NOT #statPulse.workingDone.winder[0];   // rising edge of #instJellyRollWinderLoadJob2.jobStatus.completed
   #statPulse.workingDone.winder[0] := #instJellyRollWinderLoadJob2.jobStatus.completed;
   IF #_w1 THEN "Unit1.Em7.ControlNodes".jellyRollWinder.jobInterface.loadJob2.workingDone := TRUE; END_IF;
   #_w2 := #instJellyRollWinderWinding1Job3.jobStatus.completed AND NOT #statPulse.workingDone.winder[1];   // rising edge of #instJellyRollWinderWinding1Job3.jobStatus.completed
   #statPulse.workingDone.winder[1] := #instJellyRollWinderWinding1Job3.jobStatus.completed;
   IF #_w2 THEN
       "Unit1.Em7.ControlNodes".jellyRollWinder.jobInterface.winding1Job3.workingDone := TRUE;
   END_IF;
   #_w3 := #instJellyRollWinderPusherReadyJob4.jobStatus.completed AND NOT #statPulse.workingDone.winder[2];   // rising edge of #instJellyRollWinderPusherReadyJob4.jobStatus.completed
   #statPulse.workingDone.winder[2] := #instJellyRollWinderPusherReadyJob4.jobStatus.completed;
   IF #_w3 THEN
       "Unit1.Em7.ControlNodes".jellyRollWinder.jobInterface.pusherReadyJob4.workingDone := TRUE;
   END_IF;
   #statTonTime[1].TON(IN := (NOT #statUnitStatus.specialFunctions.dryRun AND "Unit1.Em7.ControlNodes".cm.softCam.jrPusherAxisZ.waitPos.inPos AND "Unit1.Em7.ControlNodes".cmPusherRollerFwdBwd.monitoring.inHomePos) OR (#statUnitStatus.specialFunctions.dryRun AND #statUnitStatus.state.idle),
                       PT := T#1000ms);
   #_w4 := #statTonTime[1].Q AND NOT #statPulse.workingDone.winder[3];   // rising edge
   #statPulse.workingDone.winder[3] := #statTonTime[1].Q;
   IF #_w4 THEN
       "Unit1.Em7.ControlNodes".jellyRollWinder.jobInterface.pusherReadyJob4.workingDone := FALSE;
   END_IF;
   #_w5 := #instJellyRollWinderWinding2Job5.jobStatus.completed AND NOT #statPulse.workingDone.winder[4];   // rising edge of #instJellyRollWinderWinding2Job5.jobStatus.completed
   #statPulse.workingDone.winder[4] := #instJellyRollWinderWinding2Job5.jobStatus.completed;
   IF #_w5 THEN
       "Unit1.Em7.ControlNodes".jellyRollWinder.jobInterface.winding2Job5.workingDone := TRUE;
   END_IF;
   #_w6 := #instJellyRollWinderUnloadJob6.jobStatus.completed AND NOT #statPulse.workingDone.winder[5];   // rising edge of #instJellyRollWinderUnloadJob6.jobStatus.completed
   #statPulse.workingDone.winder[5] := #instJellyRollWinderUnloadJob6.jobStatus.completed;
   #_w7 := (NOT #unitStatus.specialFunctions.dryRun AND "Unit1.Em7.ControlNodes".cm.softCam.jrWinderFrontAxisY.waitPos.inPos AND "Unit1.Em7.ControlNodes".cm.softCam.jrWinderRearAxisY.waitPos.inPos AND "Unit1.Em7.ControlNodes".cmJRWinderClampTopRearUpDown.monitoring.inHomePos AND "Unit1.Em7.ControlNodes".cmJRWinderClampBtmRearUpDown.monitoring.inHomePos AND "Unit1.Em7.ControlNodes".cmJRWinderClampTopFrontUpDown.monitoring.inHomePos AND "Unit1.Em7.ControlNodes".cmJRWinderClampBtmFrontUpDown.monitoring.inHomePos) OR (#unitStatus.specialFunctions.dryRun AND #statUnitStatus.state.idle);
   #_w8 := #_w7 AND NOT #statPulse.workingDone.winder[6];   // rising edge
   #statPulse.workingDone.winder[6] := #_w7;
   IF #_w6 OR #_w8 THEN
       "Unit1.Em7.ControlNodes".jellyRollWinder.jobInterface.loadJob2.workingDone := FALSE;
       "Unit1.Em7.ControlNodes".jellyRollWinder.jobInterface.winding1Job3.workingDone := FALSE;
       "Unit1.Em7.ControlNodes".jellyRollWinder.jobInterface.pusherReadyJob4.workingDone := FALSE;
       "Unit1.Em7.ControlNodes".jellyRollWinder.jobInterface.winding2Job5.workingDone := FALSE;
   END_IF;
   "Unit1.Em7.ControlNodes".jellyRollWinder.jobInterface.unloadJob6.workingDone := #instJellyRollWinderUnloadJob6.jobStatus.completed;
   "Unit1.Em7.ControlNodes".jellyRollWinder.jobInterface.camStopSyncJob14.workingDone := #instJellyRollWinderCamStopSyncJob14.jobStatus.completed;
END_REGION

REGION Network 49: JR Winder Operation Check
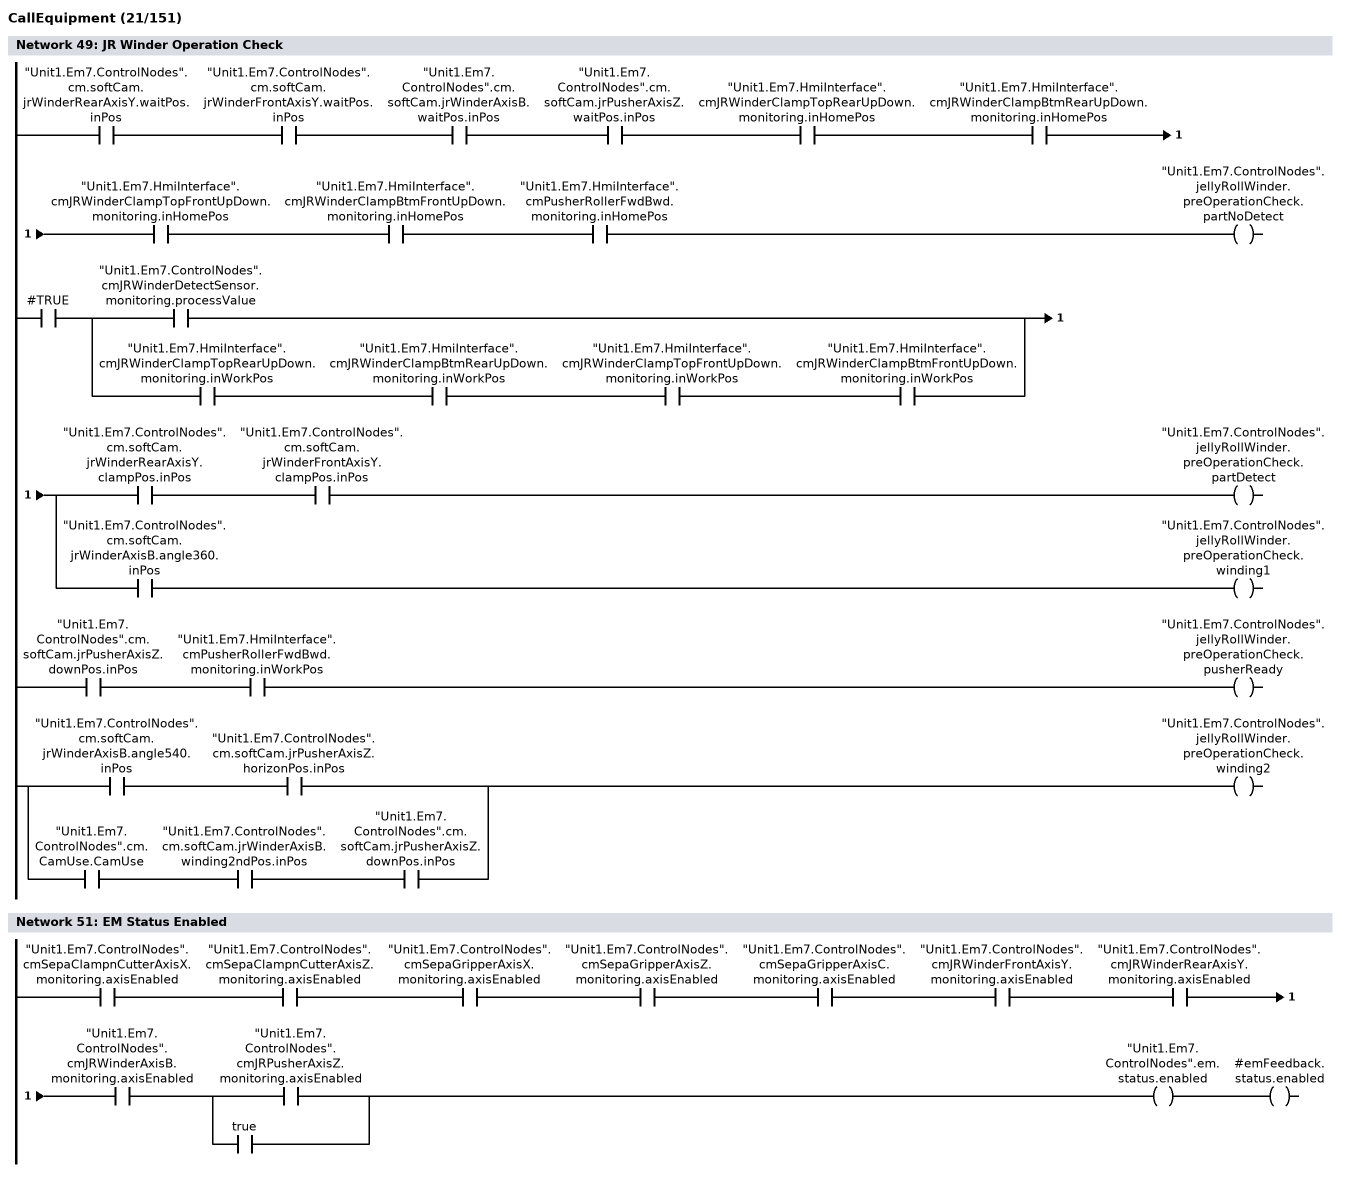
   RUNG wire#powerrail
      Contact( "Unit1.Em7.ControlNodes".cm.softCam.jrWinderRearAxisY.waitPos.inPos )
      Contact( "Unit1.Em7.ControlNodes".cm.softCam.jrWinderFrontAxisY.waitPos.inPos )
      Contact( "Unit1.Em7.ControlNodes".cm.softCam.jrWinderAxisB.waitPos.inPos )
      Contact( "Unit1.Em7.ControlNodes".cm.softCam.jrPusherAxisZ.waitPos.inPos )
      Contact( "Unit1.Em7.HmiInterface".cmJRWinderClampTopRearUpDown.monitoring.inHomePos )
      Contact( "Unit1.Em7.HmiInterface".cmJRWinderClampBtmRearUpDown.monitoring.inHomePos )
      Contact( "Unit1.Em7.HmiInterface".cmJRWinderClampTopFrontUpDown.monitoring.inHomePos )
      Contact( "Unit1.Em7.HmiInterface".cmJRWinderClampBtmFrontUpDown.monitoring.inHomePos )
      Contact( "Unit1.Em7.HmiInterface".cmPusherRollerFwdBwd.monitoring.inHomePos )
      Coil( "Unit1.Em7.ControlNodes".jellyRollWinder.preOperationCheck.partNoDetect )
   END_RUNG
   RUNG wire#powerrail
      Contact( #TRUE )
      wire#w1
      Contact( "Unit1.Em7.ControlNodes".cmJRWinderDetectSensor.monitoring.processValue )
      wire#w2
      Contact( "Unit1.Em7.ControlNodes".cm.softCam.jrWinderRearAxisY.clampPos.inPos )
      Contact( "Unit1.Em7.ControlNodes".cm.softCam.jrWinderFrontAxisY.clampPos.inPos )
      Coil( "Unit1.Em7.ControlNodes".jellyRollWinder.preOperationCheck.partDetect )
   END_RUNG
   RUNG wire#w1
      Contact( "Unit1.Em7.HmiInterface".cmJRWinderClampTopRearUpDown.monitoring.inWorkPos )
      Contact( "Unit1.Em7.HmiInterface".cmJRWinderClampBtmRearUpDown.monitoring.inWorkPos )
      Contact( "Unit1.Em7.HmiInterface".cmJRWinderClampTopFrontUpDown.monitoring.inWorkPos )
      Contact( "Unit1.Em7.HmiInterface".cmJRWinderClampBtmFrontUpDown.monitoring.inWorkPos )
   END_RUNG wire#w2
   RUNG wire#w2
      Contact( "Unit1.Em7.ControlNodes".cm.softCam.jrWinderAxisB.angle360.inPos )
      Coil( "Unit1.Em7.ControlNodes".jellyRollWinder.preOperationCheck.winding1 )
   END_RUNG
   RUNG wire#powerrail
      Contact( "Unit1.Em7.ControlNodes".cm.softCam.jrPusherAxisZ.downPos.inPos )
      Contact( "Unit1.Em7.HmiInterface".cmPusherRollerFwdBwd.monitoring.inWorkPos )
      Coil( "Unit1.Em7.ControlNodes".jellyRollWinder.preOperationCheck.pusherReady )
   END_RUNG
   RUNG wire#powerrail
      Contact( "Unit1.Em7.ControlNodes".cm.softCam.jrWinderAxisB.angle540.inPos )
      Contact( "Unit1.Em7.ControlNodes".cm.softCam.jrPusherAxisZ.horizonPos.inPos )
      wire#w3
      Coil( "Unit1.Em7.ControlNodes".jellyRollWinder.preOperationCheck.winding2 )
   END_RUNG
   RUNG wire#powerrail
      Contact( "Unit1.Em7.ControlNodes".cm.CamUse.CamUse )
      Contact( "Unit1.Em7.ControlNodes".cm.softCam.jrWinderAxisB.winding2ndPos.inPos )
      Contact( "Unit1.Em7.ControlNodes".cm.softCam.jrPusherAxisZ.downPos.inPos )
   END_RUNG wire#w3
   // the same network as SCL:
   "Unit1.Em7.ControlNodes".jellyRollWinder.preOperationCheck.partNoDetect := "Unit1.Em7.ControlNodes".cm.softCam.jrWinderRearAxisY.waitPos.inPos AND "Unit1.Em7.ControlNodes".cm.softCam.jrWinderFrontAxisY.waitPos.inPos AND "Unit1.Em7.ControlNodes".cm.softCam.jrWinderAxisB.waitPos.inPos AND "Unit1.Em7.ControlNodes".cm.softCam.jrPusherAxisZ.waitPos.inPos AND "Unit1.Em7.HmiInterface".cmJRWinderClampTopRearUpDown.monitoring.inHomePos AND "Unit1.Em7.HmiInterface".cmJRWinderClampBtmRearUpDown.monitoring.inHomePos AND "Unit1.Em7.HmiInterface".cmJRWinderClampTopFrontUpDown.monitoring.inHomePos AND "Unit1.Em7.HmiInterface".cmJRWinderClampBtmFrontUpDown.monitoring.inHomePos AND "Unit1.Em7.HmiInterface".cmPusherRollerFwdBwd.monitoring.inHomePos;
   #_w1 := #TRUE AND ("Unit1.Em7.ControlNodes".cmJRWinderDetectSensor.monitoring.processValue OR ("Unit1.Em7.HmiInterface".cmJRWinderClampTopRearUpDown.monitoring.inWorkPos AND "Unit1.Em7.HmiInterface".cmJRWinderClampBtmRearUpDown.monitoring.inWorkPos AND "Unit1.Em7.HmiInterface".cmJRWinderClampTopFrontUpDown.monitoring.inWorkPos AND "Unit1.Em7.HmiInterface".cmJRWinderClampBtmFrontUpDown.monitoring.inWorkPos));
   "Unit1.Em7.ControlNodes".jellyRollWinder.preOperationCheck.partDetect := #_w1 AND "Unit1.Em7.ControlNodes".cm.softCam.jrWinderRearAxisY.clampPos.inPos AND "Unit1.Em7.ControlNodes".cm.softCam.jrWinderFrontAxisY.clampPos.inPos;
   "Unit1.Em7.ControlNodes".jellyRollWinder.preOperationCheck.winding1 := #_w1 AND "Unit1.Em7.ControlNodes".cm.softCam.jrWinderAxisB.angle360.inPos;
   "Unit1.Em7.ControlNodes".jellyRollWinder.preOperationCheck.pusherReady := "Unit1.Em7.ControlNodes".cm.softCam.jrPusherAxisZ.downPos.inPos AND "Unit1.Em7.HmiInterface".cmPusherRollerFwdBwd.monitoring.inWorkPos;
   "Unit1.Em7.ControlNodes".jellyRollWinder.preOperationCheck.winding2 := ("Unit1.Em7.ControlNodes".cm.softCam.jrWinderAxisB.angle540.inPos AND "Unit1.Em7.ControlNodes".cm.softCam.jrPusherAxisZ.horizonPos.inPos) OR ("Unit1.Em7.ControlNodes".cm.CamUse.CamUse AND "Unit1.Em7.ControlNodes".cm.softCam.jrWinderAxisB.winding2ndPos.inPos AND "Unit1.Em7.ControlNodes".cm.softCam.jrPusherAxisZ.downPos.inPos);
END_REGION

REGION Network 51: EM Status Enabled
   RUNG wire#powerrail
      Contact( "Unit1.Em7.ControlNodes".cmSepaClampnCutterAxisX.monitoring.axisEnabled )
      Contact( "Unit1.Em7.ControlNodes".cmSepaClampnCutterAxisZ.monitoring.axisEnabled )
      Contact( "Unit1.Em7.ControlNodes".cmSepaGripperAxisX.monitoring.axisEnabled )
      Contact( "Unit1.Em7.ControlNodes".cmSepaGripperAxisZ.monitoring.axisEnabled )
      Contact( "Unit1.Em7.ControlNodes".cmSepaGripperAxisC.monitoring.axisEnabled )
      Contact( "Unit1.Em7.ControlNodes".cmJRWinderFrontAxisY.monitoring.axisEnabled )
      Contact( "Unit1.Em7.ControlNodes".cmJRWinderRearAxisY.monitoring.axisEnabled )
      Contact( "Unit1.Em7.ControlNodes".cmJRWinderAxisB.monitoring.axisEnabled )
      wire#w1
      Contact( "Unit1.Em7.ControlNodes".cmJRPusherAxisZ.monitoring.axisEnabled )
      wire#w2
      Coil( "Unit1.Em7.ControlNodes".em.status.enabled )
      Coil( #emFeedback.status.enabled )
   END_RUNG
   RUNG wire#w1
      Contact( true )
   END_RUNG wire#w2
   // the same network as SCL:
   "Unit1.Em7.ControlNodes".em.status.enabled := "Unit1.Em7.ControlNodes".cmSepaClampnCutterAxisX.monitoring.axisEnabled AND "Unit1.Em7.ControlNodes".cmSepaClampnCutterAxisZ.monitoring.axisEnabled AND "Unit1.Em7.ControlNodes".cmSepaGripperAxisX.monitoring.axisEnabled AND "Unit1.Em7.ControlNodes".cmSepaGripperAxisZ.monitoring.axisEnabled AND "Unit1.Em7.ControlNodes".cmSepaGripperAxisC.monitoring.axisEnabled AND "Unit1.Em7.ControlNodes".cmJRWinderFrontAxisY.monitoring.axisEnabled AND "Unit1.Em7.ControlNodes".cmJRWinderRearAxisY.monitoring.axisEnabled AND "Unit1.Em7.ControlNodes".cmJRWinderAxisB.monitoring.axisEnabled AND ("Unit1.Em7.ControlNodes".cmJRPusherAxisZ.monitoring.axisEnabled OR true);
   #emFeedback.status.enabled := "Unit1.Em7.ControlNodes".em.status.enabled;
END_REGION

REGION Network 52: Set EM To Initialized
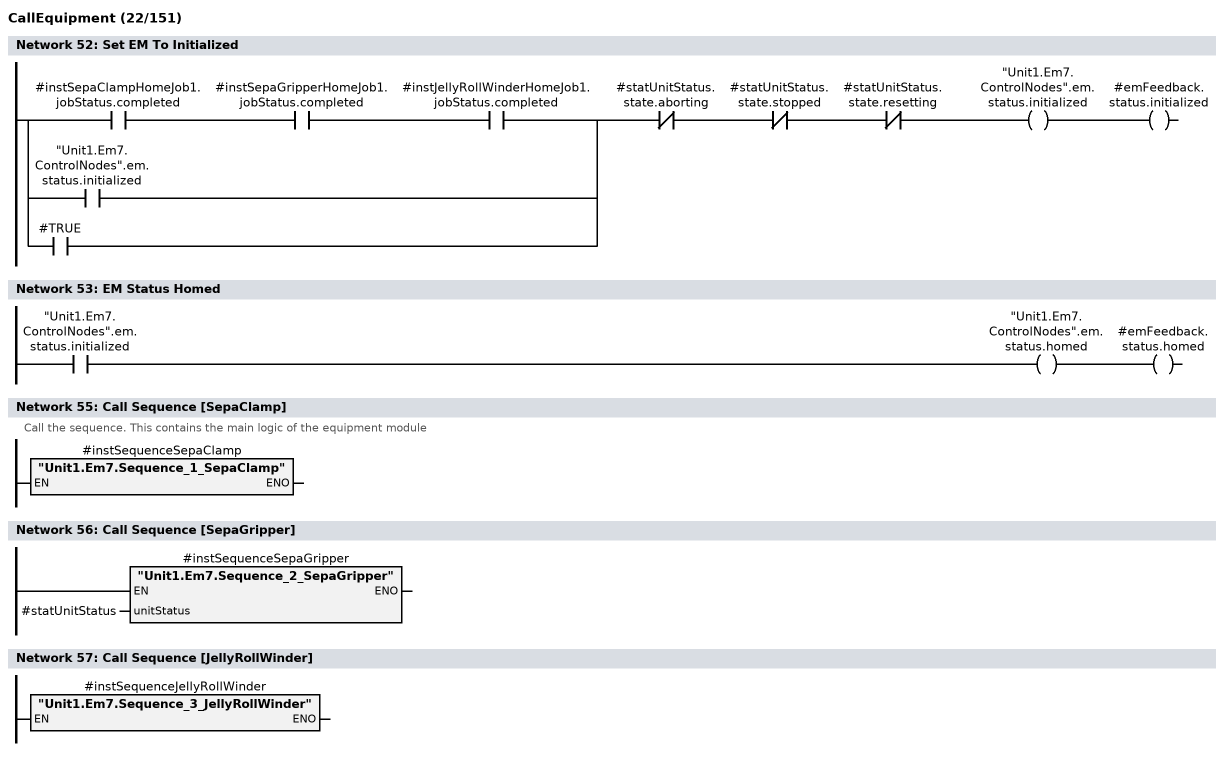
   RUNG wire#powerrail
      Contact( #instSepaClampHomeJob1.jobStatus.completed )
      Contact( #instSepaGripperHomeJob1.jobStatus.completed )
      Contact( #instJellyRollWinderHomeJob1.jobStatus.completed )
      wire#w1
      I_Contact( #statUnitStatus.state.aborting )
      I_Contact( #statUnitStatus.state.stopped )
      I_Contact( #statUnitStatus.state.resetting )
      Coil( "Unit1.Em7.ControlNodes".em.status.initialized )
      Coil( #emFeedback.status.initialized )
   END_RUNG
   RUNG wire#powerrail
      Contact( "Unit1.Em7.ControlNodes".em.status.initialized )
   END_RUNG wire#w1
   RUNG wire#powerrail
      Contact( #TRUE )
   END_RUNG wire#w1
   // the same network as SCL:
   "Unit1.Em7.ControlNodes".em.status.initialized := ((#instSepaClampHomeJob1.jobStatus.completed AND #instSepaGripperHomeJob1.jobStatus.completed AND #instJellyRollWinderHomeJob1.jobStatus.completed) OR "Unit1.Em7.ControlNodes".em.status.initialized OR #TRUE) AND NOT #statUnitStatus.state.aborting AND NOT #statUnitStatus.state.stopped AND NOT #statUnitStatus.state.resetting;
   #emFeedback.status.initialized := "Unit1.Em7.ControlNodes".em.status.initialized;
END_REGION

REGION Network 53: EM Status Homed
   RUNG wire#powerrail
      Contact( "Unit1.Em7.ControlNodes".em.status.initialized )
      Coil( "Unit1.Em7.ControlNodes".em.status.homed )
      Coil( #emFeedback.status.homed )
   END_RUNG
   // the same network as SCL:
   "Unit1.Em7.ControlNodes".em.status.homed := "Unit1.Em7.ControlNodes".em.status.initialized;
   #emFeedback.status.homed := "Unit1.Em7.ControlNodes".em.status.initialized;
END_REGION

REGION Network 55: Call Sequence [SepaClamp]
   // Call the sequence. This contains the main logic of the equipment module
   RUNG wire#powerrail
      #instSequenceSepaClamp()
   END_RUNG
   // the same network as SCL:
   #instSequenceSepaClamp();   // "Unit1.Em7.Sequence_1_SepaClamp"
END_REGION

REGION Network 56: Call Sequence [SepaGripper]
   RUNG wire#powerrail
      #instSequenceSepaGripper(unitStatus := #statUnitStatus)
   END_RUNG
   // the same network as SCL:
   #instSequenceSepaGripper(unitStatus := #statUnitStatus);   // "Unit1.Em7.Sequence_2_SepaGripper"
END_REGION

REGION Network 57: Call Sequence [JellyRollWinder]
   RUNG wire#powerrail
      #instSequenceJellyRollWinder()
   END_RUNG
   // the same network as SCL:
   #instSequenceJellyRollWinder();   // "Unit1.Em7.Sequence_3_JellyRollWinder"
END_REGION

REGION Network 58: ********** Control Modules (Axis) **********
   // Call control modules that are actuators after the em logic (jobs and sequence), so that the latest commands are applied to the actuators.
END_REGION

REGION Network 59: Reset CMS
   // Reset Axis when the unit is in the resetting state.
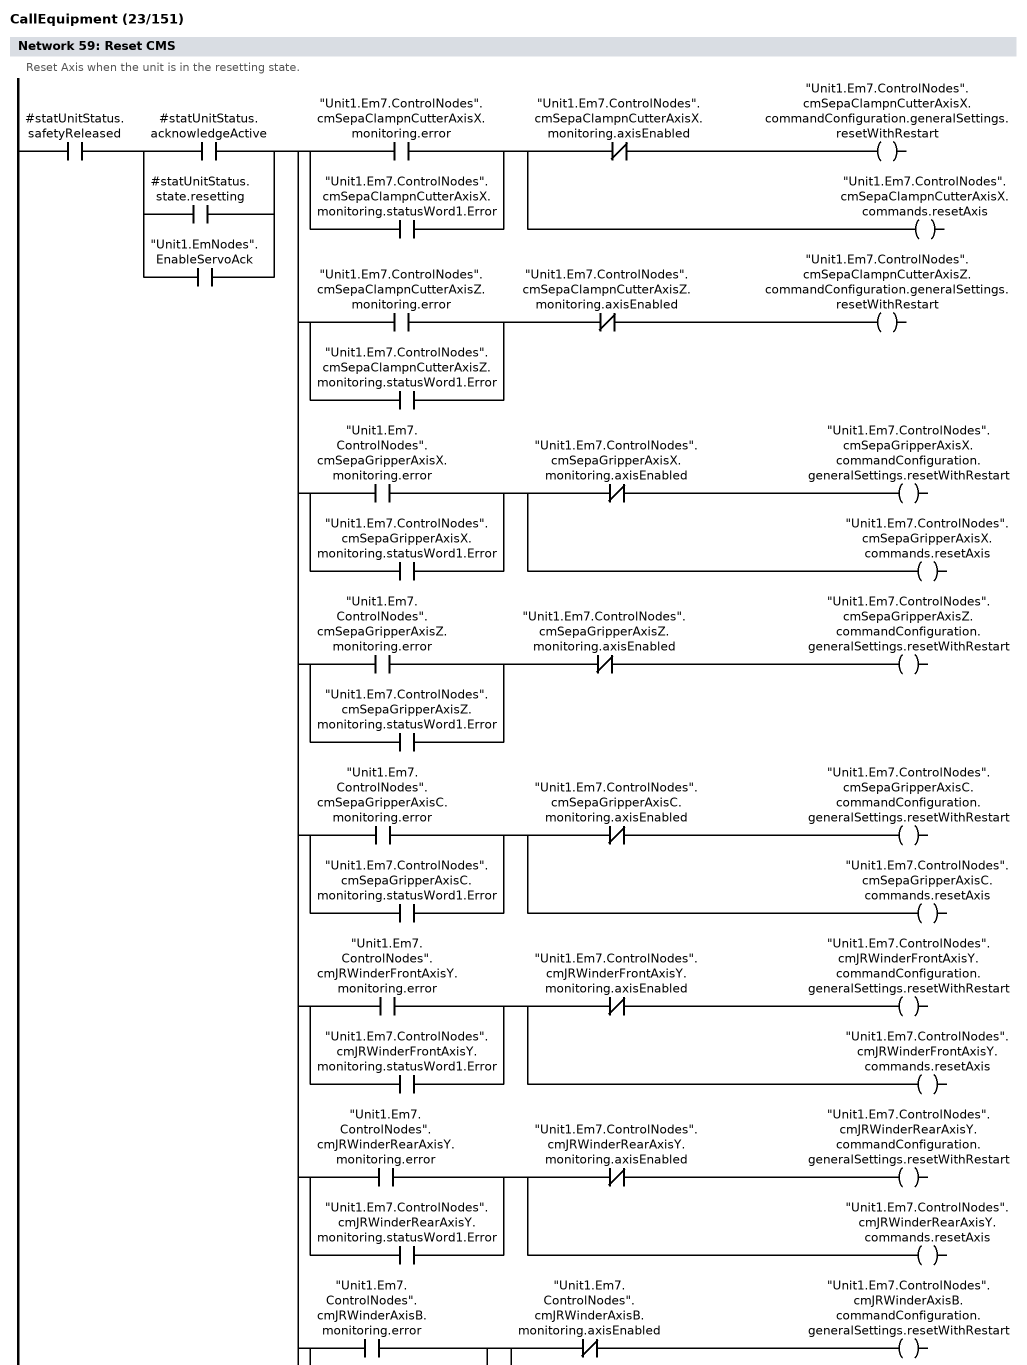
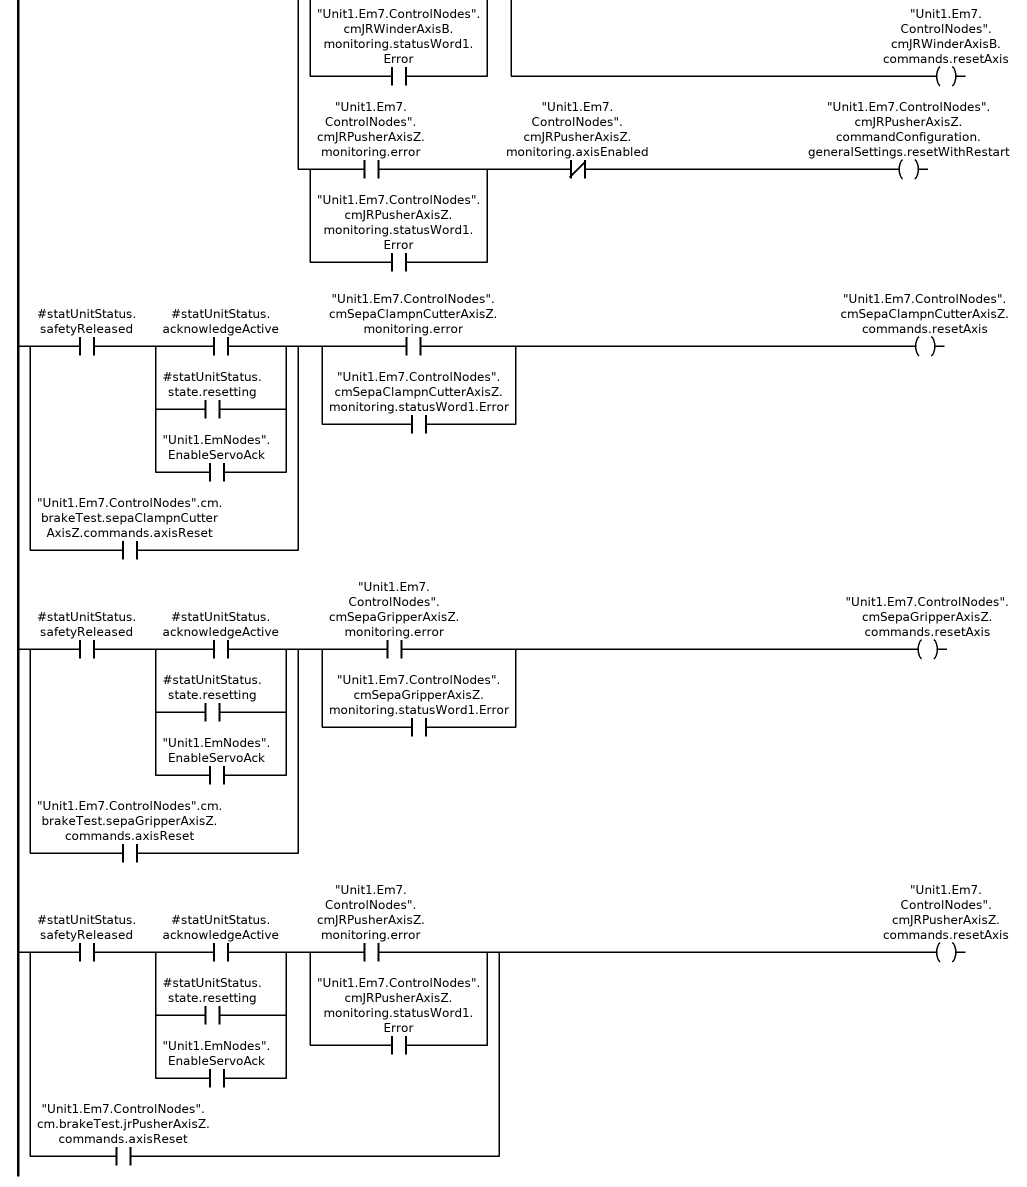
   RUNG wire#powerrail
      Contact( #statUnitStatus.safetyReleased )
      wire#w1
      Contact( #statUnitStatus.acknowledgeActive )
      wire#w2
      Contact( "Unit1.Em7.ControlNodes".cmSepaClampnCutterAxisX.monitoring.error )
      wire#w3
      I_Contact( "Unit1.Em7.ControlNodes".cmSepaClampnCutterAxisX.monitoring.axisEnabled )
      Coil( "Unit1.Em7.ControlNodes".cmSepaClampnCutterAxisX.commandConfiguration.generalSettings.resetWithRestart )
   END_RUNG
   RUNG wire#w1
      Contact( #statUnitStatus.state.resetting )
   END_RUNG wire#w2
   RUNG wire#w1
      Contact( "Unit1.EmNodes".EnableServoAck )
   END_RUNG wire#w2
   RUNG wire#w2
      Contact( "Unit1.Em7.ControlNodes".cmSepaClampnCutterAxisX.monitoring.statusWord1.Error )
   END_RUNG wire#w3
   RUNG wire#w3
      Coil( "Unit1.Em7.ControlNodes".cmSepaClampnCutterAxisX.commands.resetAxis )
   END_RUNG
   RUNG wire#w2
      Contact( "Unit1.Em7.ControlNodes".cmSepaClampnCutterAxisZ.monitoring.error )
      wire#w4
      I_Contact( "Unit1.Em7.ControlNodes".cmSepaClampnCutterAxisZ.monitoring.axisEnabled )
      Coil( "Unit1.Em7.ControlNodes".cmSepaClampnCutterAxisZ.commandConfiguration.generalSettings.resetWithRestart )
   END_RUNG
   RUNG wire#w2
      Contact( "Unit1.Em7.ControlNodes".cmSepaClampnCutterAxisZ.monitoring.statusWord1.Error )
   END_RUNG wire#w4
   RUNG wire#w2
      Contact( "Unit1.Em7.ControlNodes".cmSepaGripperAxisX.monitoring.error )
      wire#w5
      I_Contact( "Unit1.Em7.ControlNodes".cmSepaGripperAxisX.monitoring.axisEnabled )
      Coil( "Unit1.Em7.ControlNodes".cmSepaGripperAxisX.commandConfiguration.generalSettings.resetWithRestart )
   END_RUNG
   RUNG wire#w2
      Contact( "Unit1.Em7.ControlNodes".cmSepaGripperAxisX.monitoring.statusWord1.Error )
   END_RUNG wire#w5
   RUNG wire#w5
      Coil( "Unit1.Em7.ControlNodes".cmSepaGripperAxisX.commands.resetAxis )
   END_RUNG
   RUNG wire#w2
      Contact( "Unit1.Em7.ControlNodes".cmSepaGripperAxisZ.monitoring.error )
      wire#w6
      I_Contact( "Unit1.Em7.ControlNodes".cmSepaGripperAxisZ.monitoring.axisEnabled )
      Coil( "Unit1.Em7.ControlNodes".cmSepaGripperAxisZ.commandConfiguration.generalSettings.resetWithRestart )
   END_RUNG
   RUNG wire#w2
      Contact( "Unit1.Em7.ControlNodes".cmSepaGripperAxisZ.monitoring.statusWord1.Error )
   END_RUNG wire#w6
   RUNG wire#w2
      Contact( "Unit1.Em7.ControlNodes".cmSepaGripperAxisC.monitoring.error )
      wire#w7
      I_Contact( "Unit1.Em7.ControlNodes".cmSepaGripperAxisC.monitoring.axisEnabled )
      Coil( "Unit1.Em7.ControlNodes".cmSepaGripperAxisC.commandConfiguration.generalSettings.resetWithRestart )
   END_RUNG
   RUNG wire#w2
      Contact( "Unit1.Em7.ControlNodes".cmSepaGripperAxisC.monitoring.statusWord1.Error )
   END_RUNG wire#w7
   RUNG wire#w7
      Coil( "Unit1.Em7.ControlNodes".cmSepaGripperAxisC.commands.resetAxis )
   END_RUNG
   RUNG wire#w2
      Contact( "Unit1.Em7.ControlNodes".cmJRWinderFrontAxisY.monitoring.error )
      wire#w8
      I_Contact( "Unit1.Em7.ControlNodes".cmJRWinderFrontAxisY.monitoring.axisEnabled )
      Coil( "Unit1.Em7.ControlNodes".cmJRWinderFrontAxisY.commandConfiguration.generalSettings.resetWithRestart )
   END_RUNG
   RUNG wire#w2
      Contact( "Unit1.Em7.ControlNodes".cmJRWinderFrontAxisY.monitoring.statusWord1.Error )
   END_RUNG wire#w8
   RUNG wire#w8
      Coil( "Unit1.Em7.ControlNodes".cmJRWinderFrontAxisY.commands.resetAxis )
   END_RUNG
   RUNG wire#w2
      Contact( "Unit1.Em7.ControlNodes".cmJRWinderRearAxisY.monitoring.error )
      wire#w9
      I_Contact( "Unit1.Em7.ControlNodes".cmJRWinderRearAxisY.monitoring.axisEnabled )
      Coil( "Unit1.Em7.ControlNodes".cmJRWinderRearAxisY.commandConfiguration.generalSettings.resetWithRestart )
   END_RUNG
   RUNG wire#w2
      Contact( "Unit1.Em7.ControlNodes".cmJRWinderRearAxisY.monitoring.statusWord1.Error )
   END_RUNG wire#w9
   RUNG wire#w9
      Coil( "Unit1.Em7.ControlNodes".cmJRWinderRearAxisY.commands.resetAxis )
   END_RUNG
   RUNG wire#w2
      Contact( "Unit1.Em7.ControlNodes".cmJRWinderAxisB.monitoring.error )
      wire#w10
      I_Contact( "Unit1.Em7.ControlNodes".cmJRWinderAxisB.monitoring.axisEnabled )
      Coil( "Unit1.Em7.ControlNodes".cmJRWinderAxisB.commandConfiguration.generalSettings.resetWithRestart )
   END_RUNG
   RUNG wire#w2
      Contact( "Unit1.Em7.ControlNodes".cmJRWinderAxisB.monitoring.statusWord1.Error )
   END_RUNG wire#w10
   RUNG wire#w10
      Coil( "Unit1.Em7.ControlNodes".cmJRWinderAxisB.commands.resetAxis )
   END_RUNG
   RUNG wire#w2
      Contact( "Unit1.Em7.ControlNodes".cmJRPusherAxisZ.monitoring.error )
      wire#w11
      I_Contact( "Unit1.Em7.ControlNodes".cmJRPusherAxisZ.monitoring.axisEnabled )
      Coil( "Unit1.Em7.ControlNodes".cmJRPusherAxisZ.commandConfiguration.generalSettings.resetWithRestart )
   END_RUNG
   RUNG wire#w2
      Contact( "Unit1.Em7.ControlNodes".cmJRPusherAxisZ.monitoring.statusWord1.Error )
   END_RUNG wire#w11
   RUNG wire#powerrail
      Contact( #statUnitStatus.safetyReleased )
      wire#w12
      Contact( #statUnitStatus.acknowledgeActive )
      wire#w13
      Contact( "Unit1.Em7.ControlNodes".cmSepaClampnCutterAxisZ.monitoring.error )
      wire#w14
      Coil( "Unit1.Em7.ControlNodes".cmSepaClampnCutterAxisZ.commands.resetAxis )
   END_RUNG
   RUNG wire#w12
      Contact( #statUnitStatus.state.resetting )
   END_RUNG wire#w13
   RUNG wire#w12
      Contact( "Unit1.EmNodes".EnableServoAck )
   END_RUNG wire#w13
   RUNG wire#powerrail
      Contact( "Unit1.Em7.ControlNodes".cm.brakeTest.sepaClampnCutterAxisZ.commands.axisReset )
   END_RUNG wire#w13
   RUNG wire#w13
      Contact( "Unit1.Em7.ControlNodes".cmSepaClampnCutterAxisZ.monitoring.statusWord1.Error )
   END_RUNG wire#w14
   RUNG wire#powerrail
      Contact( #statUnitStatus.safetyReleased )
      wire#w15
      Contact( #statUnitStatus.acknowledgeActive )
      wire#w16
      Contact( "Unit1.Em7.ControlNodes".cmSepaGripperAxisZ.monitoring.error )
      wire#w17
      Coil( "Unit1.Em7.ControlNodes".cmSepaGripperAxisZ.commands.resetAxis )
   END_RUNG
   RUNG wire#w15
      Contact( #statUnitStatus.state.resetting )
   END_RUNG wire#w16
   RUNG wire#w15
      Contact( "Unit1.EmNodes".EnableServoAck )
   END_RUNG wire#w16
   RUNG wire#powerrail
      Contact( "Unit1.Em7.ControlNodes".cm.brakeTest.sepaGripperAxisZ.commands.axisReset )
   END_RUNG wire#w16
   RUNG wire#w16
      Contact( "Unit1.Em7.ControlNodes".cmSepaGripperAxisZ.monitoring.statusWord1.Error )
   END_RUNG wire#w17
   RUNG wire#powerrail
      Contact( #statUnitStatus.safetyReleased )
      wire#w18
      Contact( #statUnitStatus.acknowledgeActive )
      wire#w19
      Contact( "Unit1.Em7.ControlNodes".cmJRPusherAxisZ.monitoring.error )
      wire#w20
      Coil( "Unit1.Em7.ControlNodes".cmJRPusherAxisZ.commands.resetAxis )
   END_RUNG
   RUNG wire#w18
      Contact( #statUnitStatus.state.resetting )
   END_RUNG wire#w19
   RUNG wire#w18
      Contact( "Unit1.EmNodes".EnableServoAck )
   END_RUNG wire#w19
   RUNG wire#w19
      Contact( "Unit1.Em7.ControlNodes".cmJRPusherAxisZ.monitoring.statusWord1.Error )
   END_RUNG wire#w20
   RUNG wire#powerrail
      Contact( "Unit1.Em7.ControlNodes".cm.brakeTest.jrPusherAxisZ.commands.axisReset )
   END_RUNG wire#w20
   // the same network as SCL:
   #_w1 := #statUnitStatus.safetyReleased AND (#statUnitStatus.acknowledgeActive OR #statUnitStatus.state.resetting OR "Unit1.EmNodes".EnableServoAck);
   #_w2 := #_w1 AND ("Unit1.Em7.ControlNodes".cmSepaClampnCutterAxisX.monitoring.error OR "Unit1.Em7.ControlNodes".cmSepaClampnCutterAxisX.monitoring.statusWord1.Error);
   "Unit1.Em7.ControlNodes".cmSepaClampnCutterAxisX.commandConfiguration.generalSettings.resetWithRestart := #_w2 AND NOT "Unit1.Em7.ControlNodes".cmSepaClampnCutterAxisX.monitoring.axisEnabled;
   "Unit1.Em7.ControlNodes".cmSepaClampnCutterAxisX.commands.resetAxis := #_w2;
   "Unit1.Em7.ControlNodes".cmSepaClampnCutterAxisZ.commandConfiguration.generalSettings.resetWithRestart := #_w1 AND ("Unit1.Em7.ControlNodes".cmSepaClampnCutterAxisZ.monitoring.error OR "Unit1.Em7.ControlNodes".cmSepaClampnCutterAxisZ.monitoring.statusWord1.Error) AND NOT "Unit1.Em7.ControlNodes".cmSepaClampnCutterAxisZ.monitoring.axisEnabled;
   #_w3 := #_w1 AND ("Unit1.Em7.ControlNodes".cmSepaGripperAxisX.monitoring.error OR "Unit1.Em7.ControlNodes".cmSepaGripperAxisX.monitoring.statusWord1.Error);
   "Unit1.Em7.ControlNodes".cmSepaGripperAxisX.commandConfiguration.generalSettings.resetWithRestart := #_w3 AND NOT "Unit1.Em7.ControlNodes".cmSepaGripperAxisX.monitoring.axisEnabled;
   "Unit1.Em7.ControlNodes".cmSepaGripperAxisX.commands.resetAxis := #_w3;
   "Unit1.Em7.ControlNodes".cmSepaGripperAxisZ.commandConfiguration.generalSettings.resetWithRestart := #_w1 AND ("Unit1.Em7.ControlNodes".cmSepaGripperAxisZ.monitoring.error OR "Unit1.Em7.ControlNodes".cmSepaGripperAxisZ.monitoring.statusWord1.Error) AND NOT "Unit1.Em7.ControlNodes".cmSepaGripperAxisZ.monitoring.axisEnabled;
   #_w4 := #_w1 AND ("Unit1.Em7.ControlNodes".cmSepaGripperAxisC.monitoring.error OR "Unit1.Em7.ControlNodes".cmSepaGripperAxisC.monitoring.statusWord1.Error);
   "Unit1.Em7.ControlNodes".cmSepaGripperAxisC.commandConfiguration.generalSettings.resetWithRestart := #_w4 AND NOT "Unit1.Em7.ControlNodes".cmSepaGripperAxisC.monitoring.axisEnabled;
   "Unit1.Em7.ControlNodes".cmSepaGripperAxisC.commands.resetAxis := #_w4;
   #_w5 := #_w1 AND ("Unit1.Em7.ControlNodes".cmJRWinderFrontAxisY.monitoring.error OR "Unit1.Em7.ControlNodes".cmJRWinderFrontAxisY.monitoring.statusWord1.Error);
   "Unit1.Em7.ControlNodes".cmJRWinderFrontAxisY.commandConfiguration.generalSettings.resetWithRestart := #_w5 AND NOT "Unit1.Em7.ControlNodes".cmJRWinderFrontAxisY.monitoring.axisEnabled;
   "Unit1.Em7.ControlNodes".cmJRWinderFrontAxisY.commands.resetAxis := #_w5;
   #_w6 := #_w1 AND ("Unit1.Em7.ControlNodes".cmJRWinderRearAxisY.monitoring.error OR "Unit1.Em7.ControlNodes".cmJRWinderRearAxisY.monitoring.statusWord1.Error);
   "Unit1.Em7.ControlNodes".cmJRWinderRearAxisY.commandConfiguration.generalSettings.resetWithRestart := #_w6 AND NOT "Unit1.Em7.ControlNodes".cmJRWinderRearAxisY.monitoring.axisEnabled;
   "Unit1.Em7.ControlNodes".cmJRWinderRearAxisY.commands.resetAxis := #_w6;
   #_w7 := #_w1 AND ("Unit1.Em7.ControlNodes".cmJRWinderAxisB.monitoring.error OR "Unit1.Em7.ControlNodes".cmJRWinderAxisB.monitoring.statusWord1.Error);
   "Unit1.Em7.ControlNodes".cmJRWinderAxisB.commandConfiguration.generalSettings.resetWithRestart := #_w7 AND NOT "Unit1.Em7.ControlNodes".cmJRWinderAxisB.monitoring.axisEnabled;
   "Unit1.Em7.ControlNodes".cmJRWinderAxisB.commands.resetAxis := #_w7;
   "Unit1.Em7.ControlNodes".cmJRPusherAxisZ.commandConfiguration.generalSettings.resetWithRestart := #_w1 AND ("Unit1.Em7.ControlNodes".cmJRPusherAxisZ.monitoring.error OR "Unit1.Em7.ControlNodes".cmJRPusherAxisZ.monitoring.statusWord1.Error) AND NOT "Unit1.Em7.ControlNodes".cmJRPusherAxisZ.monitoring.axisEnabled;
   "Unit1.Em7.ControlNodes".cmSepaClampnCutterAxisZ.commands.resetAxis := ((#statUnitStatus.safetyReleased AND (#statUnitStatus.acknowledgeActive OR #statUnitStatus.state.resetting OR "Unit1.EmNodes".EnableServoAck)) OR "Unit1.Em7.ControlNodes".cm.brakeTest.sepaClampnCutterAxisZ.commands.axisReset) AND ("Unit1.Em7.ControlNodes".cmSepaClampnCutterAxisZ.monitoring.error OR "Unit1.Em7.ControlNodes".cmSepaClampnCutterAxisZ.monitoring.statusWord1.Error);
   "Unit1.Em7.ControlNodes".cmSepaGripperAxisZ.commands.resetAxis := ((#statUnitStatus.safetyReleased AND (#statUnitStatus.acknowledgeActive OR #statUnitStatus.state.resetting OR "Unit1.EmNodes".EnableServoAck)) OR "Unit1.Em7.ControlNodes".cm.brakeTest.sepaGripperAxisZ.commands.axisReset) AND ("Unit1.Em7.ControlNodes".cmSepaGripperAxisZ.monitoring.error OR "Unit1.Em7.ControlNodes".cmSepaGripperAxisZ.monitoring.statusWord1.Error);
   "Unit1.Em7.ControlNodes".cmJRPusherAxisZ.commands.resetAxis := (#statUnitStatus.safetyReleased AND (#statUnitStatus.acknowledgeActive OR #statUnitStatus.state.resetting OR "Unit1.EmNodes".EnableServoAck) AND ("Unit1.Em7.ControlNodes".cmJRPusherAxisZ.monitoring.error OR "Unit1.Em7.ControlNodes".cmJRPusherAxisZ.monitoring.statusWord1.Error)) OR "Unit1.Em7.ControlNodes".cm.brakeTest.jrPusherAxisZ.commands.axisReset;
END_REGION

REGION Network 60: Enable/Disable CMs
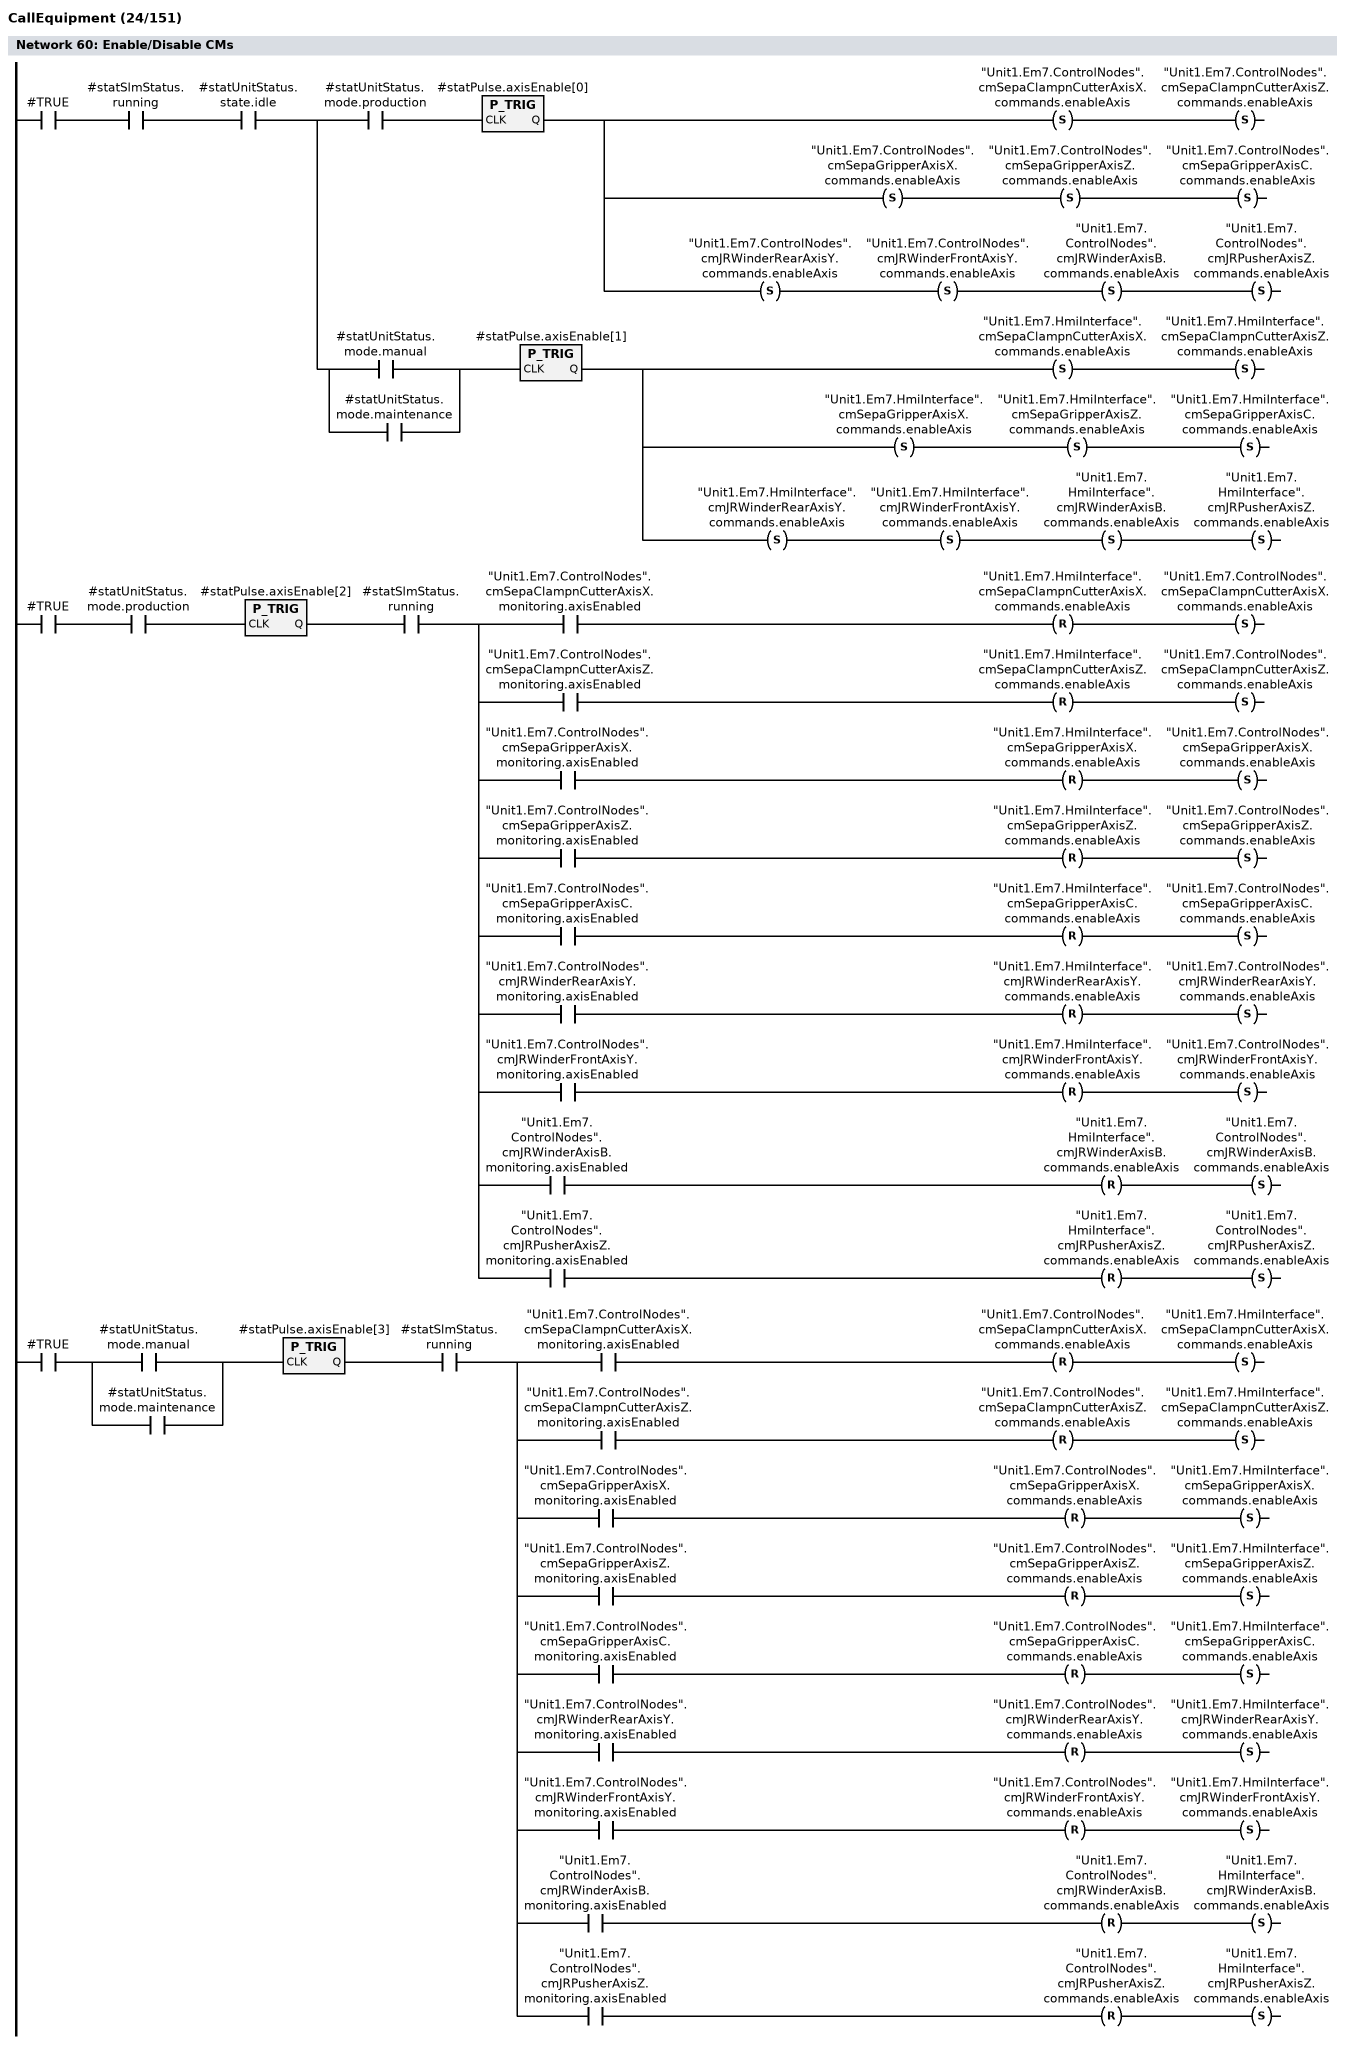
   RUNG wire#powerrail
      Contact( #TRUE )
      Contact( #statSlmStatus.running )
      Contact( #statUnitStatus.state.idle )
      wire#w1
      Contact( #statUnitStatus.mode.production )
      P_Trig( #statPulse.axisEnable[0] )
      wire#w2
      S_Coil( "Unit1.Em7.ControlNodes".cmSepaClampnCutterAxisX.commands.enableAxis )
      S_Coil( "Unit1.Em7.ControlNodes".cmSepaClampnCutterAxisZ.commands.enableAxis )
   END_RUNG
   RUNG wire#w2
      S_Coil( "Unit1.Em7.ControlNodes".cmSepaGripperAxisX.commands.enableAxis )
      S_Coil( "Unit1.Em7.ControlNodes".cmSepaGripperAxisZ.commands.enableAxis )
      S_Coil( "Unit1.Em7.ControlNodes".cmSepaGripperAxisC.commands.enableAxis )
   END_RUNG
   RUNG wire#w2
      S_Coil( "Unit1.Em7.ControlNodes".cmJRWinderRearAxisY.commands.enableAxis )
      S_Coil( "Unit1.Em7.ControlNodes".cmJRWinderFrontAxisY.commands.enableAxis )
      S_Coil( "Unit1.Em7.ControlNodes".cmJRWinderAxisB.commands.enableAxis )
      S_Coil( "Unit1.Em7.ControlNodes".cmJRPusherAxisZ.commands.enableAxis )
   END_RUNG
   RUNG wire#w1
      Contact( #statUnitStatus.mode.manual )
      wire#w3
      P_Trig( #statPulse.axisEnable[1] )
      wire#w4
      S_Coil( "Unit1.Em7.HmiInterface".cmSepaClampnCutterAxisX.commands.enableAxis )
      S_Coil( "Unit1.Em7.HmiInterface".cmSepaClampnCutterAxisZ.commands.enableAxis )
   END_RUNG
   RUNG wire#w1
      Contact( #statUnitStatus.mode.maintenance )
   END_RUNG wire#w3
   RUNG wire#w4
      S_Coil( "Unit1.Em7.HmiInterface".cmSepaGripperAxisX.commands.enableAxis )
      S_Coil( "Unit1.Em7.HmiInterface".cmSepaGripperAxisZ.commands.enableAxis )
      S_Coil( "Unit1.Em7.HmiInterface".cmSepaGripperAxisC.commands.enableAxis )
   END_RUNG
   RUNG wire#w4
      S_Coil( "Unit1.Em7.HmiInterface".cmJRWinderRearAxisY.commands.enableAxis )
      S_Coil( "Unit1.Em7.HmiInterface".cmJRWinderFrontAxisY.commands.enableAxis )
      S_Coil( "Unit1.Em7.HmiInterface".cmJRWinderAxisB.commands.enableAxis )
      S_Coil( "Unit1.Em7.HmiInterface".cmJRPusherAxisZ.commands.enableAxis )
   END_RUNG
   RUNG wire#powerrail
      Contact( #TRUE )
      Contact( #statUnitStatus.mode.production )
      P_Trig( #statPulse.axisEnable[2] )
      Contact( #statSlmStatus.running )
      wire#w5
      Contact( "Unit1.Em7.ControlNodes".cmSepaClampnCutterAxisX.monitoring.axisEnabled )
      R_Coil( "Unit1.Em7.HmiInterface".cmSepaClampnCutterAxisX.commands.enableAxis )
      S_Coil( "Unit1.Em7.ControlNodes".cmSepaClampnCutterAxisX.commands.enableAxis )
   END_RUNG
   RUNG wire#w5
      Contact( "Unit1.Em7.ControlNodes".cmSepaClampnCutterAxisZ.monitoring.axisEnabled )
      R_Coil( "Unit1.Em7.HmiInterface".cmSepaClampnCutterAxisZ.commands.enableAxis )
      S_Coil( "Unit1.Em7.ControlNodes".cmSepaClampnCutterAxisZ.commands.enableAxis )
   END_RUNG
   RUNG wire#w5
      Contact( "Unit1.Em7.ControlNodes".cmSepaGripperAxisX.monitoring.axisEnabled )
      R_Coil( "Unit1.Em7.HmiInterface".cmSepaGripperAxisX.commands.enableAxis )
      S_Coil( "Unit1.Em7.ControlNodes".cmSepaGripperAxisX.commands.enableAxis )
   END_RUNG
   RUNG wire#w5
      Contact( "Unit1.Em7.ControlNodes".cmSepaGripperAxisZ.monitoring.axisEnabled )
      R_Coil( "Unit1.Em7.HmiInterface".cmSepaGripperAxisZ.commands.enableAxis )
      S_Coil( "Unit1.Em7.ControlNodes".cmSepaGripperAxisZ.commands.enableAxis )
   END_RUNG
   RUNG wire#w5
      Contact( "Unit1.Em7.ControlNodes".cmSepaGripperAxisC.monitoring.axisEnabled )
      R_Coil( "Unit1.Em7.HmiInterface".cmSepaGripperAxisC.commands.enableAxis )
      S_Coil( "Unit1.Em7.ControlNodes".cmSepaGripperAxisC.commands.enableAxis )
   END_RUNG
   RUNG wire#w5
      Contact( "Unit1.Em7.ControlNodes".cmJRWinderRearAxisY.monitoring.axisEnabled )
      R_Coil( "Unit1.Em7.HmiInterface".cmJRWinderRearAxisY.commands.enableAxis )
      S_Coil( "Unit1.Em7.ControlNodes".cmJRWinderRearAxisY.commands.enableAxis )
   END_RUNG
   RUNG wire#w5
      Contact( "Unit1.Em7.ControlNodes".cmJRWinderFrontAxisY.monitoring.axisEnabled )
      R_Coil( "Unit1.Em7.HmiInterface".cmJRWinderFrontAxisY.commands.enableAxis )
      S_Coil( "Unit1.Em7.ControlNodes".cmJRWinderFrontAxisY.commands.enableAxis )
   END_RUNG
   RUNG wire#w5
      Contact( "Unit1.Em7.ControlNodes".cmJRWinderAxisB.monitoring.axisEnabled )
      R_Coil( "Unit1.Em7.HmiInterface".cmJRWinderAxisB.commands.enableAxis )
      S_Coil( "Unit1.Em7.ControlNodes".cmJRWinderAxisB.commands.enableAxis )
   END_RUNG
   RUNG wire#w5
      Contact( "Unit1.Em7.ControlNodes".cmJRPusherAxisZ.monitoring.axisEnabled )
      R_Coil( "Unit1.Em7.HmiInterface".cmJRPusherAxisZ.commands.enableAxis )
      S_Coil( "Unit1.Em7.ControlNodes".cmJRPusherAxisZ.commands.enableAxis )
   END_RUNG
   RUNG wire#powerrail
      Contact( #TRUE )
      wire#w6
      Contact( #statUnitStatus.mode.manual )
      wire#w7
      P_Trig( #statPulse.axisEnable[3] )
      Contact( #statSlmStatus.running )
      wire#w8
      Contact( "Unit1.Em7.ControlNodes".cmSepaClampnCutterAxisX.monitoring.axisEnabled )
      R_Coil( "Unit1.Em7.ControlNodes".cmSepaClampnCutterAxisX.commands.enableAxis )
      S_Coil( "Unit1.Em7.HmiInterface".cmSepaClampnCutterAxisX.commands.enableAxis )
   END_RUNG
   RUNG wire#w6
      Contact( #statUnitStatus.mode.maintenance )
   END_RUNG wire#w7
   RUNG wire#w8
      Contact( "Unit1.Em7.ControlNodes".cmSepaClampnCutterAxisZ.monitoring.axisEnabled )
      R_Coil( "Unit1.Em7.ControlNodes".cmSepaClampnCutterAxisZ.commands.enableAxis )
      S_Coil( "Unit1.Em7.HmiInterface".cmSepaClampnCutterAxisZ.commands.enableAxis )
   END_RUNG
   RUNG wire#w8
      Contact( "Unit1.Em7.ControlNodes".cmSepaGripperAxisX.monitoring.axisEnabled )
      R_Coil( "Unit1.Em7.ControlNodes".cmSepaGripperAxisX.commands.enableAxis )
      S_Coil( "Unit1.Em7.HmiInterface".cmSepaGripperAxisX.commands.enableAxis )
   END_RUNG
   RUNG wire#w8
      Contact( "Unit1.Em7.ControlNodes".cmSepaGripperAxisZ.monitoring.axisEnabled )
      R_Coil( "Unit1.Em7.ControlNodes".cmSepaGripperAxisZ.commands.enableAxis )
      S_Coil( "Unit1.Em7.HmiInterface".cmSepaGripperAxisZ.commands.enableAxis )
   END_RUNG
   RUNG wire#w8
      Contact( "Unit1.Em7.ControlNodes".cmSepaGripperAxisC.monitoring.axisEnabled )
      R_Coil( "Unit1.Em7.ControlNodes".cmSepaGripperAxisC.commands.enableAxis )
      S_Coil( "Unit1.Em7.HmiInterface".cmSepaGripperAxisC.commands.enableAxis )
   END_RUNG
   RUNG wire#w8
      Contact( "Unit1.Em7.ControlNodes".cmJRWinderRearAxisY.monitoring.axisEnabled )
      R_Coil( "Unit1.Em7.ControlNodes".cmJRWinderRearAxisY.commands.enableAxis )
      S_Coil( "Unit1.Em7.HmiInterface".cmJRWinderRearAxisY.commands.enableAxis )
   END_RUNG
   RUNG wire#w8
      Contact( "Unit1.Em7.ControlNodes".cmJRWinderFrontAxisY.monitoring.axisEnabled )
      R_Coil( "Unit1.Em7.ControlNodes".cmJRWinderFrontAxisY.commands.enableAxis )
      S_Coil( "Unit1.Em7.HmiInterface".cmJRWinderFrontAxisY.commands.enableAxis )
   END_RUNG
   RUNG wire#w8
      Contact( "Unit1.Em7.ControlNodes".cmJRWinderAxisB.monitoring.axisEnabled )
      R_Coil( "Unit1.Em7.ControlNodes".cmJRWinderAxisB.commands.enableAxis )
      S_Coil( "Unit1.Em7.HmiInterface".cmJRWinderAxisB.commands.enableAxis )
   END_RUNG
   RUNG wire#w8
      Contact( "Unit1.Em7.ControlNodes".cmJRPusherAxisZ.monitoring.axisEnabled )
      R_Coil( "Unit1.Em7.ControlNodes".cmJRPusherAxisZ.commands.enableAxis )
      S_Coil( "Unit1.Em7.HmiInterface".cmJRPusherAxisZ.commands.enableAxis )
   END_RUNG
   // the same network as SCL:
   #_w1 := #TRUE AND #statSlmStatus.running AND #statUnitStatus.state.idle;
   #_w2 := #_w1 AND #statUnitStatus.mode.production;
   #_w3 := #_w2 AND NOT #statPulse.axisEnable[0];   // rising edge
   #statPulse.axisEnable[0] := #_w2;
   IF #_w3 THEN
       "Unit1.Em7.ControlNodes".cmSepaClampnCutterAxisX.commands.enableAxis := TRUE;
       "Unit1.Em7.ControlNodes".cmSepaClampnCutterAxisZ.commands.enableAxis := TRUE;
       "Unit1.Em7.ControlNodes".cmSepaGripperAxisX.commands.enableAxis := TRUE;
       "Unit1.Em7.ControlNodes".cmSepaGripperAxisZ.commands.enableAxis := TRUE;
       "Unit1.Em7.ControlNodes".cmSepaGripperAxisC.commands.enableAxis := TRUE;
       "Unit1.Em7.ControlNodes".cmJRWinderRearAxisY.commands.enableAxis := TRUE;
       "Unit1.Em7.ControlNodes".cmJRWinderFrontAxisY.commands.enableAxis := TRUE;
       "Unit1.Em7.ControlNodes".cmJRWinderAxisB.commands.enableAxis := TRUE;
       "Unit1.Em7.ControlNodes".cmJRPusherAxisZ.commands.enableAxis := TRUE;
   END_IF;
   #_w4 := #_w1 AND (#statUnitStatus.mode.manual OR #statUnitStatus.mode.maintenance);
   #_w5 := #_w4 AND NOT #statPulse.axisEnable[1];   // rising edge
   #statPulse.axisEnable[1] := #_w4;
   IF #_w5 THEN
       "Unit1.Em7.HmiInterface".cmSepaClampnCutterAxisX.commands.enableAxis := TRUE;
       "Unit1.Em7.HmiInterface".cmSepaClampnCutterAxisZ.commands.enableAxis := TRUE;
       "Unit1.Em7.HmiInterface".cmSepaGripperAxisX.commands.enableAxis := TRUE;
       "Unit1.Em7.HmiInterface".cmSepaGripperAxisZ.commands.enableAxis := TRUE;
       "Unit1.Em7.HmiInterface".cmSepaGripperAxisC.commands.enableAxis := TRUE;
       "Unit1.Em7.HmiInterface".cmJRWinderRearAxisY.commands.enableAxis := TRUE;
       "Unit1.Em7.HmiInterface".cmJRWinderFrontAxisY.commands.enableAxis := TRUE;
       "Unit1.Em7.HmiInterface".cmJRWinderAxisB.commands.enableAxis := TRUE;
       "Unit1.Em7.HmiInterface".cmJRPusherAxisZ.commands.enableAxis := TRUE;
   END_IF;
   #_w6 := #TRUE AND #statUnitStatus.mode.production;
   #_w7 := #_w6 AND NOT #statPulse.axisEnable[2];   // rising edge
   #statPulse.axisEnable[2] := #_w6;
   #_w8 := #_w7 AND #statSlmStatus.running;
   IF #_w8 AND "Unit1.Em7.ControlNodes".cmSepaClampnCutterAxisX.monitoring.axisEnabled THEN
       "Unit1.Em7.HmiInterface".cmSepaClampnCutterAxisX.commands.enableAxis := FALSE;
       "Unit1.Em7.ControlNodes".cmSepaClampnCutterAxisX.commands.enableAxis := TRUE;
   END_IF;
   IF #_w8 AND "Unit1.Em7.ControlNodes".cmSepaClampnCutterAxisZ.monitoring.axisEnabled THEN
       "Unit1.Em7.HmiInterface".cmSepaClampnCutterAxisZ.commands.enableAxis := FALSE;
       "Unit1.Em7.ControlNodes".cmSepaClampnCutterAxisZ.commands.enableAxis := TRUE;
   END_IF;
   IF #_w8 AND "Unit1.Em7.ControlNodes".cmSepaGripperAxisX.monitoring.axisEnabled THEN
       "Unit1.Em7.HmiInterface".cmSepaGripperAxisX.commands.enableAxis := FALSE;
       "Unit1.Em7.ControlNodes".cmSepaGripperAxisX.commands.enableAxis := TRUE;
   END_IF;
   IF #_w8 AND "Unit1.Em7.ControlNodes".cmSepaGripperAxisZ.monitoring.axisEnabled THEN
       "Unit1.Em7.HmiInterface".cmSepaGripperAxisZ.commands.enableAxis := FALSE;
       "Unit1.Em7.ControlNodes".cmSepaGripperAxisZ.commands.enableAxis := TRUE;
   END_IF;
   IF #_w8 AND "Unit1.Em7.ControlNodes".cmSepaGripperAxisC.monitoring.axisEnabled THEN
       "Unit1.Em7.HmiInterface".cmSepaGripperAxisC.commands.enableAxis := FALSE;
       "Unit1.Em7.ControlNodes".cmSepaGripperAxisC.commands.enableAxis := TRUE;
   END_IF;
   IF #_w8 AND "Unit1.Em7.ControlNodes".cmJRWinderRearAxisY.monitoring.axisEnabled THEN
       "Unit1.Em7.HmiInterface".cmJRWinderRearAxisY.commands.enableAxis := FALSE;
       "Unit1.Em7.ControlNodes".cmJRWinderRearAxisY.commands.enableAxis := TRUE;
   END_IF;
   IF #_w8 AND "Unit1.Em7.ControlNodes".cmJRWinderFrontAxisY.monitoring.axisEnabled THEN
       "Unit1.Em7.HmiInterface".cmJRWinderFrontAxisY.commands.enableAxis := FALSE;
       "Unit1.Em7.ControlNodes".cmJRWinderFrontAxisY.commands.enableAxis := TRUE;
   END_IF;
   IF #_w8 AND "Unit1.Em7.ControlNodes".cmJRWinderAxisB.monitoring.axisEnabled THEN
       "Unit1.Em7.HmiInterface".cmJRWinderAxisB.commands.enableAxis := FALSE;
       "Unit1.Em7.ControlNodes".cmJRWinderAxisB.commands.enableAxis := TRUE;
   END_IF;
   IF #_w8 AND "Unit1.Em7.ControlNodes".cmJRPusherAxisZ.monitoring.axisEnabled THEN
       "Unit1.Em7.HmiInterface".cmJRPusherAxisZ.commands.enableAxis := FALSE;
       "Unit1.Em7.ControlNodes".cmJRPusherAxisZ.commands.enableAxis := TRUE;
   END_IF;
   #_w9 := #TRUE AND (#statUnitStatus.mode.manual OR #statUnitStatus.mode.maintenance);
   #_w10 := #_w9 AND NOT #statPulse.axisEnable[3];   // rising edge
   #statPulse.axisEnable[3] := #_w9;
   #_w11 := #_w10 AND #statSlmStatus.running;
   IF #_w11 AND "Unit1.Em7.ControlNodes".cmSepaClampnCutterAxisX.monitoring.axisEnabled THEN
       "Unit1.Em7.ControlNodes".cmSepaClampnCutterAxisX.commands.enableAxis := FALSE;
       "Unit1.Em7.HmiInterface".cmSepaClampnCutterAxisX.commands.enableAxis := TRUE;
   END_IF;
   IF #_w11 AND "Unit1.Em7.ControlNodes".cmSepaClampnCutterAxisZ.monitoring.axisEnabled THEN
       "Unit1.Em7.ControlNodes".cmSepaClampnCutterAxisZ.commands.enableAxis := FALSE;
       "Unit1.Em7.HmiInterface".cmSepaClampnCutterAxisZ.commands.enableAxis := TRUE;
   END_IF;
   IF #_w11 AND "Unit1.Em7.ControlNodes".cmSepaGripperAxisX.monitoring.axisEnabled THEN
       "Unit1.Em7.ControlNodes".cmSepaGripperAxisX.commands.enableAxis := FALSE;
       "Unit1.Em7.HmiInterface".cmSepaGripperAxisX.commands.enableAxis := TRUE;
   END_IF;
   IF #_w11 AND "Unit1.Em7.ControlNodes".cmSepaGripperAxisZ.monitoring.axisEnabled THEN
       "Unit1.Em7.ControlNodes".cmSepaGripperAxisZ.commands.enableAxis := FALSE;
       "Unit1.Em7.HmiInterface".cmSepaGripperAxisZ.commands.enableAxis := TRUE;
   END_IF;
   IF #_w11 AND "Unit1.Em7.ControlNodes".cmSepaGripperAxisC.monitoring.axisEnabled THEN
       "Unit1.Em7.ControlNodes".cmSepaGripperAxisC.commands.enableAxis := FALSE;
       "Unit1.Em7.HmiInterface".cmSepaGripperAxisC.commands.enableAxis := TRUE;
   END_IF;
   IF #_w11 AND "Unit1.Em7.ControlNodes".cmJRWinderRearAxisY.monitoring.axisEnabled THEN
       "Unit1.Em7.ControlNodes".cmJRWinderRearAxisY.commands.enableAxis := FALSE;
       "Unit1.Em7.HmiInterface".cmJRWinderRearAxisY.commands.enableAxis := TRUE;
   END_IF;
   IF #_w11 AND "Unit1.Em7.ControlNodes".cmJRWinderFrontAxisY.monitoring.axisEnabled THEN
       "Unit1.Em7.ControlNodes".cmJRWinderFrontAxisY.commands.enableAxis := FALSE;
       "Unit1.Em7.HmiInterface".cmJRWinderFrontAxisY.commands.enableAxis := TRUE;
   END_IF;
   IF #_w11 AND "Unit1.Em7.ControlNodes".cmJRWinderAxisB.monitoring.axisEnabled THEN
       "Unit1.Em7.ControlNodes".cmJRWinderAxisB.commands.enableAxis := FALSE;
       "Unit1.Em7.HmiInterface".cmJRWinderAxisB.commands.enableAxis := TRUE;
   END_IF;
   IF #_w11 AND "Unit1.Em7.ControlNodes".cmJRPusherAxisZ.monitoring.axisEnabled THEN
       "Unit1.Em7.ControlNodes".cmJRPusherAxisZ.commands.enableAxis := FALSE;
       "Unit1.Em7.HmiInterface".cmJRPusherAxisZ.commands.enableAxis := TRUE;
   END_IF;
END_REGION

